LIN {X 0,Y 314.203,Z 248.248,A -85,B 0,C 180,E1 -15768.607,E2 -15768.607} C_VEL
LIN {X 0,Y 312.569,Z 240.551,A -85,B 0,C 180,E1 -15771.085,E2 -15771.085} C_VEL
LIN {X 0,Y 312.557,Z 240.551,A -85,B 0,C 180,E1 -15775.292,E2 -15775.292} C_VEL
LIN {X 0,Y 312.526,Z 240.558,A -85,B 0,C 180,E1 -15778.714,E2 -15778.714} C_VEL
LIN {X 0,Y 312.503,Z 240.561,A -85,B 0,C 180,E1 -15782.666,E2 -15782.666} C_VEL
LIN {X 0,Y 312.507,Z 240.552,A -85,B 0,C 180,E1 -15786.781,E2 -15786.781} C_VEL
LIN {X 0,Y 311.84,Z 240.639,A -85,B 0,C 180,E1 -15787.857,E2 -15787.857} C_VEL
LIN {X 0,Y 308.958,Z 240.997,A -85,B 0,C 180,E1 -15789.608,E2 -15789.608} C_VEL
LIN {X 0,Y 306.532,Z 241.301,A -85,B 0,C 180,E1 -15791.029,E2 -15791.029} C_VEL
LIN {X 0,Y 305.522,Z 241.426,A -85,B 0,C 180,E1 -15792.129,E2 -15792.129} C_VEL
LIN {X 0,Y 305.456,Z 241.437,A -85,B 0,C 180,E1 -15792.502,E2 -15792.502} C_VEL
LIN {X 0,Y 305.443,Z 241.437,A -85,B 0,C 180,E1 -15796.348,E2 -15796.348} C_VEL
LIN {X 0,Y 305.459,Z 241.433,A -85,B 0,C 180,E1 -15799.892,E2 -15799.892} C_VEL
LIN {X 0,Y 305.481,Z 241.43,A -85,B 0,C 180,E1 -15803.632,E2 -15803.632} C_VEL
LIN {X 0,Y 305.466,Z 241.432,A -85,B 0,C 180,E1 -15806.483,E2 -15806.483} C_VEL
LIN {X 0,Y 305.459,Z 241.43,A -85,B 0,C 180,E1 -15809.59,E2 -15809.59} C_VEL
LIN {X 0,Y 305.516,Z 241.431,A -85,B 0,C 180,E1 -15812.608,E2 -15812.608} C_VEL
LIN {X 0,Y 305.509,Z 241.423,A -85,B 0,C 180,E1 -15815.539,E2 -15815.539} C_VEL
LIN {X 0,Y 305.521,Z 241.42,A -85,B 0,C 180,E1 -15819.815,E2 -15819.815} C_VEL
LIN {X 0,Y 305.575,Z 241.422,A -85,B 0,C 180,E1 -15822.603,E2 -15822.603} C_VEL
LIN {X 0,Y 305.65,Z 241.406,A -85,B 0,C 180,E1 -15825.349,E2 -15825.349} C_VEL
LIN {X 0,Y 305.625,Z 241.402,A -85,B 0,C 180,E1 -15829.399,E2 -15829.399} C_VEL
LIN {X 0,Y 305.749,Z 241.393,A -85,B 0,C 180,E1 -15832.073,E2 -15832.073} C_VEL
LIN {X 0,Y 305.674,Z 241.41,A -85,B 0,C 180,E1 -15834.723,E2 -15834.723} C_VEL
LIN {X 0,Y 305.954,Z 241.374,A -85,B 0,C 180,E1 -15838.684,E2 -15838.684} C_VEL
LIN {X 0,Y 305.955,Z 241.371,A -85,B 0,C 180,E1 -15841.316,E2 -15841.316} C_VEL
LIN {X 0,Y 305.853,Z 241.389,A -85,B 0,C 180,E1 -15846.597,E2 -15846.597} C_VEL
LIN {X 0,Y 305.736,Z 241.397,A -85,B 0,C 180,E1 -15849.26,E2 -15849.26} C_VEL
LIN {X 0,Y 305.587,Z 241.416,A -85,B 0,C 180,E1 -15853.296,E2 -15853.296} C_VEL
LIN {X 0,Y 305.551,Z 241.422,A -85,B 0,C 180,E1 -15856.022,E2 -15856.022} C_VEL
LIN {X 0,Y 305.485,Z 241.429,A -85,B 0,C 180,E1 -15860.187,E2 -15860.187} C_VEL
LIN {X 0,Y 305.487,Z 241.432,A -85,B 0,C 180,E1 -15864.463,E2 -15864.463} C_VEL
LIN {X 0,Y 305.467,Z 241.432,A -85,B 0,C 180,E1 -15867.397,E2 -15867.397} C_VEL
LIN {X 0,Y 305.433,Z 241.438,A -85,B 0,C 180,E1 -15870.412,E2 -15870.412} C_VEL
LIN {X 0,Y 305.465,Z 241.434,A -85,B 0,C 180,E1 -15874.078,E2 -15874.078} C_VEL
LIN {X 0,Y 305.469,Z 241.436,A -85,B 0,C 180,E1 -15876.74,E2 -15876.74} C_VEL
LIN {X 0,Y 305.409,Z 241.444,A -85,B 0,C 180,E1 -15880.59,E2 -15880.59} C_VEL
LIN {X 0,Y 305.422,Z 241.438,A -85,B 0,C 180,E1 -15883.656,E2 -15883.656} C_VEL
LIN {X 0,Y 305.454,Z 241.432,A -85,B 0,C 180,E1 -15887.414,E2 -15887.414} C_VEL
LIN {X 0,Y 305.477,Z 241.431,A -85,B 0,C 180,E1 -15891.598,E2 -15891.598} C_VEL
LIN {X 0,Y 305.463,Z 241.436,A -85,B 0,C 180,E1 -15894.887,E2 -15894.887} C_VEL
LIN {X 0,Y 305.481,Z 241.475,A -85,B 0,C 180,E1 -15898.346,E2 -15898.346} C_VEL
LIN {X 0,Y 308.107,Z 253.691,A -85,B 0,C 180,E1 -15902.12,E2 -15902.12} C_VEL
LIN {X 0,Y 309.418,Z 261.563,A -85,B 0,C 180,E1 -15904.434,E2 -15904.434} C_VEL
LIN {X 0,Y 309.266,Z 263.81,A -85,B 0,C 180,E1 -15905.048,E2 -15905.048} C_VEL
LIN {X 0,Y 313.254,Z 289.715,A -85,B 0,C 180,E1 -15905.992,E2 -15905.992} C_VEL
LIN {X 0,Y 315.292,Z 305.062,A -85,B 0,C 180,E1 -15906.504,E2 -15906.504} C_VEL
LIN {X 0,Y 313.764,Z 372.606,A -85,B 0,C 180,E1 -15908.051,E2 -15908.051} C_VEL
LIN {X 0,Y 312.937,Z 386.537,A -85,B 0,C 180,E1 -15908.639,E2 -15908.639} C_VEL
LIN {X 0,Y 311.957,Z 398.459,A -85,B 0,C 180,E1 -15909.39,E2 -15909.39} C_VEL
LIN {X 0,Y 310.802,Z 409.719,A -85,B 0,C 180,E1 -15910.345,E2 -15910.345} C_VEL
LIN {X 0,Y 309.44,Z 421.391,A -85,B 0,C 180,E1 -15911.631,E2 -15911.631} C_VEL
LIN {X 0,Y 308.14,Z 431.519,A -85,B 0,C 180,E1 -15913.036,E2 -15913.036} C_VEL
LIN {X 0,Y 306.995,Z 441.335,A -85,B 0,C 180,E1 -15914.736,E2 -15914.736} C_VEL
LIN {X 0,Y 305.751,Z 450.436,A -85,B 0,C 180,E1 -15916.711,E2 -15916.711} C_VEL
LIN {X 0,Y 304.82,Z 457.766,A -85,B 0,C 180,E1 -15918.698,E2 -15918.698} C_VEL
LIN {X 0,Y 304.223,Z 463.634,A -85,B 0,C 180,E1 -15920.694,E2 -15920.694} C_VEL
LIN {X 0,Y 303.838,Z 468.245,A -85,B 0,C 180,E1 -15922.691,E2 -15922.691} C_VEL
LIN {X 0,Y 303.637,Z 471.745,A -85,B 0,C 180,E1 -15924.688,E2 -15924.688} C_VEL
LIN {X 0,Y 303.633,Z 473.5,A -85,B 0,C 180,E1 -15926.018,E2 -15926.018} C_VEL
LIN {X 0,Y 303.608,Z 474.831,A -85,B 0,C 180,E1 -15927.347,E2 -15927.347} C_VEL
LIN {X 0,Y 303.575,Z 475.764,A -85,B 0,C 180,E1 -15928.673,E2 -15928.673} C_VEL
LIN {X 0,Y 303.604,Z 476.304,A -85,B 0,C 180,E1 -15930,E2 -15930} C_VEL
LIN {X 0,Y 303.565,Z 476.407,A -85,B 0,C 180,E1 -15931.327,E2 -15931.327} C_VEL
LIN {X 0,Y 303.601,Z 476.119,A -85,B 0,C 180,E1 -15932.654,E2 -15932.654} C_VEL
LIN {X 0,Y 303.596,Z 475.445,A -85,B 0,C 180,E1 -15933.982,E2 -15933.982} C_VEL
LIN {X 0,Y 303.695,Z 473.996,A -85,B 0,C 180,E1 -15935.679,E2 -15935.679} C_VEL
LIN {X 0,Y 304.005,Z 470.949,A -85,B 0,C 180,E1 -15937.973,E2 -15937.973} C_VEL
LIN {X 0,Y 304.564,Z 467.224,A -85,B 0,C 180,E1 -15939.966,E2 -15939.966} C_VEL
LIN {X 0,Y 305.367,Z 462.397,A -85,B 0,C 180,E1 -15941.955,E2 -15941.955} C_VEL
LIN {X 0,Y 306.595,Z 456.323,A -85,B 0,C 180,E1 -15943.927,E2 -15943.927} C_VEL
LIN {X 0,Y 308.09,Z 448.786,A -85,B 0,C 180,E1 -15945.887,E2 -15945.887} C_VEL
LIN {X 0,Y 309.541,Z 441.029,A -85,B 0,C 180,E1 -15947.523,E2 -15947.523} C_VEL
LIN {X 0,Y 311.171,Z 431.759,A -85,B 0,C 180,E1 -15949.117,E2 -15949.117} C_VEL
LIN {X 0,Y 313.02,Z 421.391,A -85,B 0,C 180,E1 -15950.537,E2 -15950.537} C_VEL
LIN {X 0,Y 314.798,Z 409.893,A -85,B 0,C 180,E1 -15951.787,E2 -15951.787} C_VEL
LIN {X 0,Y 316.426,Z 397.786,A -85,B 0,C 180,E1 -15952.786,E2 -15952.786} C_VEL
LIN {X 0,Y 317.74,Z 384.331,A -85,B 0,C 180,E1 -15953.591,E2 -15953.591} C_VEL
LIN {X 0,Y 318.583,Z 371.861,A -85,B 0,C 180,E1 -15954.086,E2 -15954.086} C_VEL
LIN {X 0,Y 320.398,Z 307.143,A -85,B 0,C 180,E1 -15955.554,E2 -15955.554} C_VEL
LIN {X 0,Y 317.446,Z 289.422,A -85,B 0,C 180,E1 -15956.282,E2 -15956.282} C_VEL
LIN {X 0,Y 313.767,Z 271.603,A -85,B 0,C 180,E1 -15957.106,E2 -15957.106} C_VEL
LIN {X 0,Y 310.5,Z 263.435,A -85,B 0,C 180,E1 -15957.679,E2 -15957.679} C_VEL
LIN {X 0,Y 308.691,Z 254.815,A -85,B 0,C 180,E1 -15960.435,E2 -15960.435} C_VEL
LIN {X 0,Y 306.228,Z 244.486,A -85,B 0,C 180,E1 -15963.93,E2 -15963.93} C_VEL
LIN {X 0,Y 305.497,Z 241.428,A -85,B 0,C 180,E1 -15965.04,E2 -15965.04} C_VEL
LIN {X 0,Y 305.441,Z 241.438,A -85,B 0,C 180,E1 -15968.527,E2 -15968.527} C_VEL
LIN {X 0,Y 305.455,Z 241.437,A -85,B 0,C 180,E1 -15972.586,E2 -15972.586} C_VEL
LIN {X 0,Y 305.422,Z 241.44,A -85,B 0,C 180,E1 -15976.344,E2 -15976.344} C_VEL
LIN {X 0,Y 305.41,Z 241.442,A -85,B 0,C 180,E1 -15979.885,E2 -15979.885} C_VEL
LIN {X 0,Y 305.463,Z 241.43,A -85,B 0,C 180,E1 -15983.636,E2 -15983.636} C_VEL
LIN {X 0,Y 305.465,Z 241.426,A -85,B 0,C 180,E1 -15986.483,E2 -15986.483} C_VEL
LIN {X 0,Y 305.435,Z 241.433,A -85,B 0,C 180,E1 -15989.588,E2 -15989.588} C_VEL
LIN {X 0,Y 305.472,Z 241.433,A -85,B 0,C 180,E1 -15992.604,E2 -15992.604} C_VEL
LIN {X 0,Y 305.489,Z 241.428,A -85,B 0,C 180,E1 -15995.537,E2 -15995.537} C_VEL
LIN {X 0,Y 305.496,Z 241.428,A -85,B 0,C 180,E1 -15999.814,E2 -15999.814} C_VEL
LIN {X 0,Y 305.545,Z 241.42,A -85,B 0,C 180,E1 -16002.601,E2 -16002.601} C_VEL
LIN {X 0,Y 305.628,Z 241.415,A -85,B 0,C 180,E1 -16005.348,E2 -16005.348} C_VEL
LIN {X 0,Y 305.639,Z 241.408,A -85,B 0,C 180,E1 -16009.4,E2 -16009.4} C_VEL
LIN {X 0,Y 305.81,Z 241.384,A -85,B 0,C 180,E1 -16012.074,E2 -16012.074} C_VEL
LIN {X 0,Y 305.682,Z 241.404,A -85,B 0,C 180,E1 -16014.723,E2 -16014.723} C_VEL
LIN {X 0,Y 305.953,Z 241.364,A -85,B 0,C 180,E1 -16018.684,E2 -16018.684} C_VEL
LIN {X 0,Y 305.954,Z 241.373,A -85,B 0,C 180,E1 -16021.316,E2 -16021.316} C_VEL
LIN {X 0,Y 305.672,Z 241.408,A -85,B 0,C 180,E1 -16025.277,E2 -16025.277} C_VEL
LIN {X 0,Y 305.752,Z 241.388,A -85,B 0,C 180,E1 -16027.927,E2 -16027.927} C_VEL
LIN {X 0,Y 305.6,Z 241.414,A -85,B 0,C 180,E1 -16031.945,E2 -16031.945} C_VEL
LIN {X 0,Y 305.61,Z 241.413,A -85,B 0,C 180,E1 -16035.015,E2 -16035.015} C_VEL
LIN {X 0,Y 305.563,Z 241.418,A -85,B 0,C 180,E1 -16039.437,E2 -16039.437} C_VEL
LIN {X 0,Y 305.492,Z 241.422,A -85,B 0,C 180,E1 -16043.041,E2 -16043.041} C_VEL
LIN {X 0,Y 305.527,Z 241.418,A -85,B 0,C 180,E1 -16046.219,E2 -16046.219} C_VEL
LIN {X 0,Y 305.49,Z 241.432,A -85,B 0,C 180,E1 -16049.048,E2 -16049.048} C_VEL
LIN {X 0,Y 305.444,Z 241.437,A -85,B 0,C 180,E1 -16051.952,E2 -16051.952} C_VEL
LIN {X 0,Y 305.464,Z 241.437,A -85,B 0,C 180,E1 -16055.113,E2 -16055.113} C_VEL
LIN {X 0,Y 305.469,Z 241.433,A -85,B 0,C 180,E1 -16058.533,E2 -16058.533} C_VEL
LIN {X 0,Y 305.46,Z 241.436,A -85,B 0,C 180,E1 -16062.587,E2 -16062.587} C_VEL
LIN {X 0,Y 305.441,Z 241.431,A -85,B 0,C 180,E1 -16066.348,E2 -16066.348} C_VEL
LIN {X 0,Y 305.411,Z 241.44,A -85,B 0,C 180,E1 -16069.885,E2 -16069.885} C_VEL
LIN {X 0,Y 305.486,Z 241.455,A -85,B 0,C 180,E1 -16073.384,E2 -16073.384} C_VEL
LIN {X 0,Y 307.289,Z 248.962,A -85,B 0,C 180,E1 -16076.037,E2 -16076.037} C_VEL
LIN {X 0,Y 315.614,Z 266.974,A -85,B 0,C 180,E1 -16077.391,E2 -16077.391} C_VEL
LIN {X 0,Y 319.918,Z 277.771,A -85,B 0,C 180,E1 -16078.094,E2 -16078.094} C_VEL
LIN {X 0,Y 321.078,Z 283.904,A -85,B 0,C 180,E1 -16078.36,E2 -16078.36} C_VEL
LIN {X 0,Y 318.96,Z 356.614,A -85,B 0,C 180,E1 -16080.007,E2 -16080.007} C_VEL
LIN {X 0,Y 318.074,Z 370.586,A -85,B 0,C 180,E1 -16080.598,E2 -16080.598} C_VEL
LIN {X 0,Y 316.992,Z 382.524,A -85,B 0,C 180,E1 -16081.351,E2 -16081.351} C_VEL
LIN {X 0,Y 315.553,Z 393.762,A -85,B 0,C 180,E1 -16082.294,E2 -16082.294} C_VEL
LIN {X 0,Y 313.929,Z 405.364,A -85,B 0,C 180,E1 -16083.572,E2 -16083.572} C_VEL
LIN {X 0,Y 312.157,Z 415.883,A -85,B 0,C 180,E1 -16085.03,E2 -16085.03} C_VEL
LIN {X 0,Y 310.4,Z 425.242,A -85,B 0,C 180,E1 -16086.657,E2 -16086.657} C_VEL
LIN {X 0,Y 308.671,Z 434.282,A -85,B 0,C 180,E1 -16088.636,E2 -16088.636} C_VEL
LIN {X 0,Y 307.202,Z 441.538,A -85,B 0,C 180,E1 -16090.627,E2 -16090.627} C_VEL
LIN {X 0,Y 305.99,Z 447.301,A -85,B 0,C 180,E1 -16092.627,E2 -16092.627} C_VEL
LIN {X 0,Y 305.111,Z 451.814,A -85,B 0,C 180,E1 -16094.639,E2 -16094.639} C_VEL
LIN {X 0,Y 304.426,Z 455.23,A -85,B 0,C 180,E1 -16096.652,E2 -16096.652} C_VEL
LIN {X 0,Y 304.065,Z 456.919,A -85,B 0,C 180,E1 -16097.994,E2 -16097.994} C_VEL
LIN {X 0,Y 303.653,Z 459.087,A -85,B 0,C 180,E1 -16100.676,E2 -16100.676} C_VEL
LIN {X 0,Y 303.619,Z 459.549,A -85,B 0,C 180,E1 -16102.017,E2 -16102.017} C_VEL
LIN {X 0,Y 303.622,Z 459.352,A -85,B 0,C 180,E1 -16104.464,E2 -16104.464} C_VEL
LIN {X 0,Y 303.648,Z 458.56,A -85,B 0,C 180,E1 -16106.018,E2 -16106.018} C_VEL
LIN {X 0,Y 303.661,Z 457.434,A -85,B 0,C 180,E1 -16107.347,E2 -16107.347} C_VEL
LIN {X 0,Y 303.935,Z 453.917,A -85,B 0,C 180,E1 -16110,E2 -16110} C_VEL
LIN {X 0,Y 304.323,Z 450.115,A -85,B 0,C 180,E1 -16111.985,E2 -16111.985} C_VEL
LIN {X 0,Y 304.901,Z 445.198,A -85,B 0,C 180,E1 -16113.965,E2 -16113.965} C_VEL
LIN {X 0,Y 305.66,Z 439.023,A -85,B 0,C 180,E1 -16115.939,E2 -16115.939} C_VEL
LIN {X 0,Y 306.784,Z 431.306,A -85,B 0,C 180,E1 -16117.9,E2 -16117.9} C_VEL
LIN {X 0,Y 308.173,Z 421.655,A -85,B 0,C 180,E1 -16119.848,E2 -16119.848} C_VEL
LIN {X 0,Y 309.434,Z 411.687,A -85,B 0,C 180,E1 -16121.463,E2 -16121.463} C_VEL
LIN {X 0,Y 310.732,Z 400.394,A -85,B 0,C 180,E1 -16122.906,E2 -16122.906} C_VEL
LIN {X 0,Y 311.868,Z 389.33,A -85,B 0,C 180,E1 -16124.02,E2 -16124.02} C_VEL
LIN {X 0,Y 312.948,Z 376.702,A -85,B 0,C 180,E1 -16124.986,E2 -16124.986} C_VEL
LIN {X 0,Y 313.662,Z 363.863,A -85,B 0,C 180,E1 -16125.681,E2 -16125.681} C_VEL
LIN {X 0,Y 314.124,Z 351.155,A -85,B 0,C 180,E1 -16126.115,E2 -16126.115} C_VEL
LIN {X 0,Y 315.815,Z 279.626,A -85,B 0,C 180,E1 -16127.715,E2 -16127.715} C_VEL
LIN {X 0,Y 312.921,Z 264.379,A -85,B 0,C 180,E1 -16128.293,E2 -16128.293} C_VEL
LIN {X 0,Y 307.038,Z 248.411,A -85,B 0,C 180,E1 -16129.163,E2 -16129.163} C_VEL
LIN {X 0,Y 305.523,Z 241.427,A -85,B 0,C 180,E1 -16131.507,E2 -16131.507} C_VEL
LIN {X 0,Y 305.51,Z 241.428,A -85,B 0,C 180,E1 -16135.918,E2 -16135.918} C_VEL
LIN {X 0,Y 305.465,Z 241.435,A -85,B 0,C 180,E1 -16139.039,E2 -16139.039} C_VEL
LIN {X 0,Y 305.439,Z 241.436,A -85,B 0,C 180,E1 -16141.953,E2 -16141.953} C_VEL
LIN {X 0,Y 305.464,Z 241.434,A -85,B 0,C 180,E1 -16145.113,E2 -16145.113} C_VEL
LIN {X 0,Y 305.451,Z 241.438,A -85,B 0,C 180,E1 -16148.529,E2 -16148.529} C_VEL
LIN {X 0,Y 305.456,Z 241.437,A -85,B 0,C 180,E1 -16152.502,E2 -16152.502} C_VEL
LIN {X 0,Y 304.819,Z 241.522,A -85,B 0,C 180,E1 -16153.601,E2 -16153.601} C_VEL
LIN {X 0,Y 301.929,Z 241.878,A -85,B 0,C 180,E1 -16155.388,E2 -16155.388} C_VEL
LIN {X 0,Y 299.469,Z 242.183,A -85,B 0,C 180,E1 -16156.839,E2 -16156.839} C_VEL
LIN {X 0,Y 298.435,Z 242.308,A -85,B 0,C 180,E1 -16157.963,E2 -16157.963} C_VEL
LIN {X 0,Y 298.365,Z 242.318,A -85,B 0,C 180,E1 -16158.344,E2 -16158.344} C_VEL
LIN {X 0,Y 298.409,Z 242.312,A -85,B 0,C 180,E1 -16162.241,E2 -16162.241} C_VEL
LIN {X 0,Y 298.409,Z 242.309,A -85,B 0,C 180,E1 -16165.581,E2 -16165.581} C_VEL
LIN {X 0,Y 298.393,Z 242.31,A -85,B 0,C 180,E1 -16168.791,E2 -16168.791} C_VEL
LIN {X 0,Y 298.458,Z 242.305,A -85,B 0,C 180,E1 -16171.903,E2 -16171.903} C_VEL
LIN {X 0,Y 298.484,Z 242.3,A -85,B 0,C 180,E1 -16174.924,E2 -16174.924} C_VEL
LIN {X 0,Y 298.451,Z 242.301,A -85,B 0,C 180,E1 -16179.315,E2 -16179.315} C_VEL
LIN {X 0,Y 298.539,Z 242.295,A -85,B 0,C 180,E1 -16182.179,E2 -16182.179} C_VEL
LIN {X 0,Y 298.594,Z 242.286,A -85,B 0,C 180,E1 -16184.995,E2 -16184.995} C_VEL
LIN {X 0,Y 298.584,Z 242.279,A -85,B 0,C 180,E1 -16189.146,E2 -16189.146} C_VEL
LIN {X 0,Y 298.7,Z 242.27,A -85,B 0,C 180,E1 -16191.884,E2 -16191.884} C_VEL
LIN {X 0,Y 298.642,Z 242.286,A -85,B 0,C 180,E1 -16194.598,E2 -16194.598} C_VEL
LIN {X 0,Y 298.921,Z 242.249,A -85,B 0,C 180,E1 -16198.653,E2 -16198.653} C_VEL
LIN {X 0,Y 298.922,Z 242.247,A -85,B 0,C 180,E1 -16201.347,E2 -16201.347} C_VEL
LIN {X 0,Y 298.798,Z 242.267,A -85,B 0,C 180,E1 -16206.754,E2 -16206.754} C_VEL
LIN {X 0,Y 298.681,Z 242.275,A -85,B 0,C 180,E1 -16209.48,E2 -16209.48} C_VEL
LIN {X 0,Y 298.546,Z 242.293,A -85,B 0,C 180,E1 -16213.616,E2 -16213.616} C_VEL
LIN {X 0,Y 298.484,Z 242.305,A -85,B 0,C 180,E1 -16216.412,E2 -16216.412} C_VEL
LIN {X 0,Y 298.46,Z 242.302,A -85,B 0,C 180,E1 -16219.627,E2 -16219.627} C_VEL
LIN {X 0,Y 298.424,Z 242.308,A -85,B 0,C 180,E1 -16223.6,E2 -16223.6} C_VEL
LIN {X 0,Y 298.413,Z 242.314,A -85,B 0,C 180,E1 -16226.582,E2 -16226.582} C_VEL
LIN {X 0,Y 298.398,Z 242.311,A -85,B 0,C 180,E1 -16229.643,E2 -16229.643} C_VEL
LIN {X 0,Y 298.392,Z 242.316,A -85,B 0,C 180,E1 -16232.801,E2 -16232.801} C_VEL
LIN {X 0,Y 298.442,Z 242.31,A -85,B 0,C 180,E1 -16236.806,E2 -16236.806} C_VEL
LIN {X 0,Y 298.348,Z 242.32,A -85,B 0,C 180,E1 -16241.079,E2 -16241.079} C_VEL
LIN {X 0,Y 298.399,Z 242.314,A -85,B 0,C 180,E1 -16243.103,E2 -16243.103} C_VEL
LIN {X 0,Y 298.403,Z 242.312,A -85,B 0,C 180,E1 -16246.921,E2 -16246.921} C_VEL
LIN {X 0,Y 298.404,Z 242.313,A -85,B 0,C 180,E1 -16251.006,E2 -16251.006} C_VEL
LIN {X 0,Y 298.433,Z 242.31,A -85,B 0,C 180,E1 -16253.932,E2 -16253.932} C_VEL
LIN {X 0,Y 298.433,Z 242.519,A -85,B 0,C 180,E1 -16257.972,E2 -16257.972} C_VEL
LIN {X 0,Y 300.775,Z 253.216,A -85,B 0,C 180,E1 -16261.379,E2 -16261.379} C_VEL
LIN {X 0,Y 302.428,Z 262.577,A -85,B 0,C 180,E1 -16264.216,E2 -16264.216} C_VEL
LIN {X 0,Y 302.48,Z 263.631,A -85,B 0,C 180,E1 -16264.521,E2 -16264.521} C_VEL
LIN {X 0,Y 306.547,Z 289.629,A -85,B 0,C 180,E1 -16265.498,E2 -16265.498} C_VEL
LIN {X 0,Y 308.645,Z 305.97,A -85,B 0,C 180,E1 -16266.055,E2 -16266.055} C_VEL
LIN {X 0,Y 307.12,Z 371.987,A -85,B 0,C 180,E1 -16267.595,E2 -16267.595} C_VEL
LIN {X 0,Y 306.318,Z 385.292,A -85,B 0,C 180,E1 -16268.154,E2 -16268.154} C_VEL
LIN {X 0,Y 305.322,Z 397.489,A -85,B 0,C 180,E1 -16268.921,E2 -16268.921} C_VEL
LIN {X 0,Y 304.095,Z 408.965,A -85,B 0,C 180,E1 -16269.893,E2 -16269.893} C_VEL
LIN {X 0,Y 302.674,Z 420.748,A -85,B 0,C 180,E1 -16271.206,E2 -16271.206} C_VEL
LIN {X 0,Y 301.271,Z 431.211,A -85,B 0,C 180,E1 -16272.679,E2 -16272.679} C_VEL
LIN {X 0,Y 300.124,Z 440.854,A -85,B 0,C 180,E1 -16274.378,E2 -16274.378} C_VEL
LIN {X 0,Y 298.819,Z 450.007,A -85,B 0,C 180,E1 -16276.397,E2 -16276.397} C_VEL
LIN {X 0,Y 297.807,Z 457.377,A -85,B 0,C 180,E1 -16278.428,E2 -16278.428} C_VEL
LIN {X 0,Y 297.195,Z 463.286,A -85,B 0,C 180,E1 -16280.472,E2 -16280.472} C_VEL
LIN {X 0,Y 296.785,Z 467.932,A -85,B 0,C 180,E1 -16282.516,E2 -16282.516} C_VEL
LIN {X 0,Y 296.552,Z 471.46,A -85,B 0,C 180,E1 -16284.56,E2 -16284.56} C_VEL
LIN {X 0,Y 296.531,Z 473.241,A -85,B 0,C 180,E1 -16285.923,E2 -16285.923} C_VEL
LIN {X 0,Y 296.534,Z 474.588,A -85,B 0,C 180,E1 -16287.283,E2 -16287.283} C_VEL
LIN {X 0,Y 296.494,Z 475.534,A -85,B 0,C 180,E1 -16288.642,E2 -16288.642} C_VEL
LIN {X 0,Y 296.518,Z 476.092,A -85,B 0,C 180,E1 -16290,E2 -16290} C_VEL
LIN {X 0,Y 296.485,Z 476.218,A -85,B 0,C 180,E1 -16291.358,E2 -16291.358} C_VEL
LIN {X 0,Y 296.526,Z 475.943,A -85,B 0,C 180,E1 -16292.717,E2 -16292.717} C_VEL
LIN {X 0,Y 296.554,Z 474.235,A -85,B 0,C 180,E1 -16295.44,E2 -16295.44} C_VEL
LIN {X 0,Y 296.694,Z 472.757,A -85,B 0,C 180,E1 -16296.802,E2 -16296.802} C_VEL
LIN {X 0,Y 297.109,Z 469.75,A -85,B 0,C 180,E1 -16298.845,E2 -16298.845} C_VEL
LIN {X 0,Y 297.806,Z 465.703,A -85,B 0,C 180,E1 -16300.882,E2 -16300.882} C_VEL
LIN {X 0,Y 298.943,Z 459.502,A -85,B 0,C 180,E1 -16303.251,E2 -16303.251} C_VEL
LIN {X 0,Y 300.491,Z 452.767,A -85,B 0,C 180,E1 -16305.255,E2 -16305.255} C_VEL
LIN {X 0,Y 302.131,Z 444.475,A -85,B 0,C 180,E1 -16307.241,E2 -16307.241} C_VEL
LIN {X 0,Y 303.7,Z 435.852,A -85,B 0,C 180,E1 -16308.904,E2 -16308.904} C_VEL
LIN {X 0,Y 305.745,Z 425.298,A -85,B 0,C 180,E1 -16310.521,E2 -16310.521} C_VEL
LIN {X 0,Y 307.497,Z 414.847,A -85,B 0,C 180,E1 -16311.802,E2 -16311.802} C_VEL
LIN {X 0,Y 309.257,Z 403.325,A -85,B 0,C 180,E1 -16312.903,E2 -16312.903} C_VEL
LIN {X 0,Y 310.698,Z 391.377,A -85,B 0,C 180,E1 -16313.761,E2 -16313.761} C_VEL
LIN {X 0,Y 311.845,Z 378.463,A -85,B 0,C 180,E1 -16314.419,E2 -16314.419} C_VEL
LIN {X 0,Y 312.563,Z 366.37,A -85,B 0,C 180,E1 -16314.802,E2 -16314.802} C_VEL
LIN {X 0,Y 314.036,Z 306.607,A -85,B 0,C 180,E1 -16316.181,E2 -16316.181} C_VEL
LIN {X 0,Y 309.092,Z 279.498,A -85,B 0,C 180,E1 -16317.388,E2 -16317.388} C_VEL
LIN {X 0,Y 307.454,Z 273.208,A -85,B 0,C 180,E1 -16317.728,E2 -16317.728} C_VEL
LIN {X 0,Y 303.263,Z 263.264,A -85,B 0,C 180,E1 -16318.458,E2 -16318.458} C_VEL
LIN {X 0,Y 301.198,Z 253.595,A -85,B 0,C 180,E1 -16321.669,E2 -16321.669} C_VEL
LIN {X 0,Y 298.447,Z 242.339,A -85,B 0,C 180,E1 -16325.667,E2 -16325.667} C_VEL
LIN {X 0,Y 298.401,Z 242.316,A -85,B 0,C 180,E1 -16329.487,E2 -16329.487} C_VEL
LIN {X 0,Y 298.399,Z 242.316,A -85,B 0,C 180,E1 -16333.103,E2 -16333.103} C_VEL
LIN {X 0,Y 298.372,Z 242.32,A -85,B 0,C 180,E1 -16336.915,E2 -16336.915} C_VEL
LIN {X 0,Y 298.385,Z 242.316,A -85,B 0,C 180,E1 -16341.011,E2 -16341.011} C_VEL
LIN {X 0,Y 298.405,Z 242.311,A -85,B 0,C 180,E1 -16343.928,E2 -16343.928} C_VEL
LIN {X 0,Y 298.393,Z 242.308,A -85,B 0,C 180,E1 -16347.2,E2 -16347.2} C_VEL
LIN {X 0,Y 298.411,Z 242.303,A -85,B 0,C 180,E1 -16350.622,E2 -16350.622} C_VEL
LIN {X 0,Y 298.45,Z 242.3,A -85,B 0,C 180,E1 -16354.921,E2 -16354.921} C_VEL
LIN {X 0,Y 298.43,Z 242.304,A -85,B 0,C 180,E1 -16359.314,E2 -16359.314} C_VEL
LIN {X 0,Y 298.506,Z 242.297,A -85,B 0,C 180,E1 -16362.177,E2 -16362.177} C_VEL
LIN {X 0,Y 298.586,Z 242.289,A -85,B 0,C 180,E1 -16364.994,E2 -16364.994} C_VEL
LIN {X 0,Y 298.594,Z 242.283,A -85,B 0,C 180,E1 -16369.147,E2 -16369.147} C_VEL
LIN {X 0,Y 298.756,Z 242.263,A -85,B 0,C 180,E1 -16371.886,E2 -16371.886} C_VEL
LIN {X 0,Y 298.653,Z 242.279,A -85,B 0,C 180,E1 -16374.599,E2 -16374.599} C_VEL
LIN {X 0,Y 298.919,Z 242.24,A -85,B 0,C 180,E1 -16378.653,E2 -16378.653} C_VEL
LIN {X 0,Y 298.921,Z 242.248,A -85,B 0,C 180,E1 -16381.347,E2 -16381.347} C_VEL
LIN {X 0,Y 298.712,Z 242.273,A -85,B 0,C 180,E1 -16386.513,E2 -16386.513} C_VEL
LIN {X 0,Y 298.627,Z 242.281,A -85,B 0,C 180,E1 -16389.482,E2 -16389.482} C_VEL
LIN {X 0,Y 298.546,Z 242.287,A -85,B 0,C 180,E1 -16393.616,E2 -16393.616} C_VEL
LIN {X 0,Y 298.488,Z 242.301,A -85,B 0,C 180,E1 -16396.412,E2 -16396.412} C_VEL
LIN {X 0,Y 298.5,Z 242.3,A -85,B 0,C 180,E1 -16399.648,E2 -16399.648} C_VEL
LIN {X 0,Y 298.459,Z 242.303,A -85,B 0,C 180,E1 -16403.598,E2 -16403.598} C_VEL
LIN {X 0,Y 298.486,Z 242.294,A -85,B 0,C 180,E1 -16406.575,E2 -16406.575} C_VEL
LIN {X 0,Y 298.418,Z 242.307,A -85,B 0,C 180,E1 -16409.642,E2 -16409.642} C_VEL
LIN {X 0,Y 298.396,Z 242.314,A -85,B 0,C 180,E1 -16412.8,E2 -16412.8} C_VEL
LIN {X 0,Y 298.466,Z 242.302,A -85,B 0,C 180,E1 -16416.812,E2 -16416.812} C_VEL
LIN {X 0,Y 298.389,Z 242.315,A -85,B 0,C 180,E1 -16421.088,E2 -16421.088} C_VEL
LIN {X 0,Y 298.39,Z 242.32,A -85,B 0,C 180,E1 -16425.042,E2 -16425.042} C_VEL
LIN {X 0,Y 298.351,Z 242.328,A -85,B 0,C 180,E1 -16428.733,E2 -16428.733} C_VEL
LIN {X 0,Y 298.452,Z 242.491,A -85,B 0,C 180,E1 -16432.778,E2 -16432.778} C_VEL
LIN {X 0,Y 300.129,Z 249.165,A -85,B 0,C 180,E1 -16435.227,E2 -16435.227} C_VEL
LIN {X 0,Y 309.605,Z 269.427,A -85,B 0,C 180,E1 -16436.829,E2 -16436.829} C_VEL
LIN {X 0,Y 313.908,Z 280.009,A -85,B 0,C 180,E1 -16437.552,E2 -16437.552} C_VEL
LIN {X 0,Y 314.781,Z 284.041,A -85,B 0,C 180,E1 -16437.744,E2 -16437.744} C_VEL
LIN {X 0,Y 312.631,Z 356.824,A -85,B 0,C 180,E1 -16439.428,E2 -16439.428} C_VEL
LIN {X 0,Y 311.72,Z 370.794,A -85,B 0,C 180,E1 -16440.031,E2 -16440.031} C_VEL
LIN {X 0,Y 310.575,Z 382.725,A -85,B 0,C 180,E1 -16440.795,E2 -16440.795} C_VEL
LIN {X 0,Y 308.994,Z 394.764,A -85,B 0,C 180,E1 -16441.839,E2 -16441.839} C_VEL
LIN {X 0,Y 307.329,Z 405.969,A -85,B 0,C 180,E1 -16443.108,E2 -16443.108} C_VEL
LIN {X 0,Y 305.445,Z 416.607,A -85,B 0,C 180,E1 -16444.625,E2 -16444.625} C_VEL
LIN {X 0,Y 303.783,Z 425.029,A -85,B 0,C 180,E1 -16446.118,E2 -16446.118} C_VEL
LIN {X 0,Y 301.949,Z 434.139,A -85,B 0,C 180,E1 -16448.136,E2 -16448.136} C_VEL
LIN {X 0,Y 300.395,Z 441.456,A -85,B 0,C 180,E1 -16450.169,E2 -16450.169} C_VEL
LIN {X 0,Y 299.111,Z 447.287,A -85,B 0,C 180,E1 -16452.215,E2 -16452.215} C_VEL
LIN {X 0,Y 298.166,Z 451.853,A -85,B 0,C 180,E1 -16454.272,E2 -16454.272} C_VEL
LIN {X 0,Y 297.44,Z 455.31,A -85,B 0,C 180,E1 -16456.333,E2 -16456.333} C_VEL
LIN {X 0,Y 297.051,Z 457.026,A -85,B 0,C 180,E1 -16457.706,E2 -16457.706} C_VEL
LIN {X 0,Y 296.573,Z 459.235,A -85,B 0,C 180,E1 -16460.451,E2 -16460.451} C_VEL
LIN {X 0,Y 296.524,Z 459.736,A -85,B 0,C 180,E1 -16461.824,E2 -16461.824} C_VEL
LIN {X 0,Y 296.548,Z 459.522,A -85,B 0,C 180,E1 -16464.491,E2 -16464.491} C_VEL
LIN {X 0,Y 296.542,Z 458.807,A -85,B 0,C 180,E1 -16465.923,E2 -16465.923} C_VEL
LIN {X 0,Y 296.583,Z 457.718,A -85,B 0,C 180,E1 -16467.284,E2 -16467.284} C_VEL
LIN {X 0,Y 296.834,Z 454.246,A -85,B 0,C 180,E1 -16470,E2 -16470} C_VEL
LIN {X 0,Y 297.261,Z 450.487,A -85,B 0,C 180,E1 -16472.032,E2 -16472.032} C_VEL
LIN {X 0,Y 297.841,Z 445.618,A -85,B 0,C 180,E1 -16474.059,E2 -16474.059} C_VEL
LIN {X 0,Y 298.64,Z 439.493,A -85,B 0,C 180,E1 -16476.079,E2 -16476.079} C_VEL
LIN {X 0,Y 299.772,Z 431.868,A -85,B 0,C 180,E1 -16478.086,E2 -16478.086} C_VEL
LIN {X 0,Y 301.214,Z 422.29,A -85,B 0,C 180,E1 -16480.078,E2 -16480.078} C_VEL
LIN {X 0,Y 302.506,Z 412.426,A -85,B 0,C 180,E1 -16481.729,E2 -16481.729} C_VEL
LIN {X 0,Y 303.877,Z 401.291,A -85,B 0,C 180,E1 -16483.202,E2 -16483.202} C_VEL
LIN {X 0,Y 305.031,Z 390.396,A -85,B 0,C 180,E1 -16484.34,E2 -16484.34} C_VEL
LIN {X 0,Y 306.165,Z 378.076,A -85,B 0,C 180,E1 -16485.326,E2 -16485.326} C_VEL
LIN {X 0,Y 306.92,Z 364.959,A -85,B 0,C 180,E1 -16486.077,E2 -16486.077} C_VEL
LIN {X 0,Y 307.423,Z 352.82,A -85,B 0,C 180,E1 -16486.519,E2 -16486.519} C_VEL
LIN {X 0,Y 309.104,Z 279.856,A -85,B 0,C 180,E1 -16488.198,E2 -16488.198} C_VEL
LIN {X 0,Y 306.686,Z 267.023,A -85,B 0,C 180,E1 -16488.699,E2 -16488.699} C_VEL
LIN {X 0,Y 299.865,Z 248.66,A -85,B 0,C 180,E1 -16489.724,E2 -16489.724} C_VEL
LIN {X 0,Y 298.441,Z 242.309,A -85,B 0,C 180,E1 -16491.862,E2 -16491.862} C_VEL
LIN {X 0,Y 298.452,Z 242.309,A -85,B 0,C 180,E1 -16495.079,E2 -16495.079} C_VEL
LIN {X 0,Y 298.412,Z 242.312,A -85,B 0,C 180,E1 -16499.378,E2 -16499.378} C_VEL
LIN {X 0,Y 298.394,Z 242.317,A -85,B 0,C 180,E1 -16502.8,E2 -16502.8} C_VEL
LIN {X 0,Y 298.448,Z 242.31,A -85,B 0,C 180,E1 -16506.807,E2 -16506.807} C_VEL
LIN {X 0,Y 298.389,Z 242.315,A -85,B 0,C 180,E1 -16511.088,E2 -16511.088} C_VEL
LIN {X 0,Y 298.39,Z 242.316,A -85,B 0,C 180,E1 -16515.041,E2 -16515.041} C_VEL
LIN {X 0,Y 298.365,Z 242.318,A -85,B 0,C 180,E1 -16518.344,E2 -16518.344} C_VEL
LIN {X 0,Y 297.729,Z 242.401,A -85,B 0,C 180,E1 -16519.47,E2 -16519.47} C_VEL
LIN {X 0,Y 294.877,Z 242.754,A -85,B 0,C 180,E1 -16521.304,E2 -16521.304} C_VEL
LIN {X 0,Y 292.45,Z 243.058,A -85,B 0,C 180,E1 -16522.792,E2 -16522.792} C_VEL
LIN {X 0,Y 291.424,Z 243.182,A -85,B 0,C 180,E1 -16523.945,E2 -16523.945} C_VEL
LIN {X 0,Y 291.351,Z 243.191,A -85,B 0,C 180,E1 -16524.335,E2 -16524.335} C_VEL
LIN {X 0,Y 291.371,Z 243.178,A -85,B 0,C 180,E1 -16527.95,E2 -16527.95} C_VEL
LIN {X 0,Y 291.378,Z 243.188,A -85,B 0,C 180,E1 -16531.158,E2 -16531.158} C_VEL
LIN {X 0,Y 291.414,Z 243.184,A -85,B 0,C 180,E1 -16534.271,E2 -16534.271} C_VEL
LIN {X 0,Y 291.382,Z 243.173,A -85,B 0,C 180,E1 -16537.299,E2 -16537.299} C_VEL
LIN {X 0,Y 291.459,Z 243.173,A -85,B 0,C 180,E1 -16540.27,E2 -16540.27} C_VEL
LIN {X 0,Y 291.556,Z 243.166,A -85,B 0,C 180,E1 -16544.624,E2 -16544.624} C_VEL
LIN {X 0,Y 291.53,Z 243.156,A -85,B 0,C 180,E1 -16548.88,E2 -16548.88} C_VEL
LIN {X 0,Y 291.653,Z 243.147,A -85,B 0,C 180,E1 -16551.687,E2 -16551.687} C_VEL
LIN {X 0,Y 291.61,Z 243.16,A -85,B 0,C 180,E1 -16554.468,E2 -16554.468} C_VEL
LIN {X 0,Y 291.888,Z 243.124,A -85,B 0,C 180,E1 -16558.62,E2 -16558.62} C_VEL
LIN {X 0,Y 291.888,Z 243.123,A -85,B 0,C 180,E1 -16561.38,E2 -16561.38} C_VEL
LIN {X 0,Y 291.747,Z 243.144,A -85,B 0,C 180,E1 -16566.918,E2 -16566.918} C_VEL
LIN {X 0,Y 291.63,Z 243.153,A -85,B 0,C 180,E1 -16569.712,E2 -16569.712} C_VEL
LIN {X 0,Y 291.516,Z 243.17,A -85,B 0,C 180,E1 -16573.95,E2 -16573.95} C_VEL
LIN {X 0,Y 291.429,Z 243.181,A -85,B 0,C 180,E1 -16576.821,E2 -16576.821} C_VEL
LIN {X 0,Y 291.424,Z 243.179,A -85,B 0,C 180,E1 -16579.86,E2 -16579.86} C_VEL
LIN {X 0,Y 291.365,Z 243.189,A -85,B 0,C 180,E1 -16584.208,E2 -16584.208} C_VEL
LIN {X 0,Y 291.359,Z 243.19,A -85,B 0,C 180,E1 -16587.278,E2 -16587.278} C_VEL
LIN {X 0,Y 291.32,Z 243.195,A -85,B 0,C 180,E1 -16590.439,E2 -16590.439} C_VEL
LIN {X 0,Y 291.344,Z 243.191,A -85,B 0,C 180,E1 -16593.698,E2 -16593.698} C_VEL
LIN {X 0,Y 291.368,Z 243.189,A -85,B 0,C 180,E1 -16597.252,E2 -16597.252} C_VEL
LIN {X 0,Y 291.3,Z 243.201,A -85,B 0,C 180,E1 -16600.648,E2 -16600.648} C_VEL
LIN {X 0,Y 291.291,Z 243.202,A -85,B 0,C 180,E1 -16604.402,E2 -16604.402} C_VEL
LIN {X 0,Y 291.326,Z 243.192,A -85,B 0,C 180,E1 -16608.404,E2 -16608.404} C_VEL
LIN {X 0,Y 291.354,Z 243.191,A -85,B 0,C 180,E1 -16611.159,E2 -16611.159} C_VEL
LIN {X 0,Y 291.386,Z 243.191,A -85,B 0,C 180,E1 -16614.63,E2 -16614.63} C_VEL
LIN {X 0,Y 291.364,Z 243.198,A -85,B 0,C 180,E1 -16617.462,E2 -16617.462} C_VEL
LIN {X 0,Y 293.74,Z 254.053,A -85,B 0,C 180,E1 -16621.02,E2 -16621.02} C_VEL
LIN {X 0,Y 295.446,Z 263.563,A -85,B 0,C 180,E1 -16623.958,E2 -16623.958} C_VEL
LIN {X 0,Y 296.941,Z 270.938,A -85,B 0,C 180,E1 -16624.272,E2 -16624.272} C_VEL
LIN {X 0,Y 301.135,Z 299.015,A -85,B 0,C 180,E1 -16625.322,E2 -16625.322} C_VEL
LIN {X 0,Y 302.03,Z 307.217,A -85,B 0,C 180,E1 -16625.596,E2 -16625.596} C_VEL
LIN {X 0,Y 300.434,Z 372.513,A -85,B 0,C 180,E1 -16627.159,E2 -16627.159} C_VEL
LIN {X 0,Y 299.552,Z 386.345,A -85,B 0,C 180,E1 -16627.77,E2 -16627.77} C_VEL
LIN {X 0,Y 298.45,Z 398.742,A -85,B 0,C 180,E1 -16628.593,E2 -16628.593} C_VEL
LIN {X 0,Y 296.998,Z 411.417,A -85,B 0,C 180,E1 -16629.752,E2 -16629.752} C_VEL
LIN {X 0,Y 295.556,Z 422.706,A -85,B 0,C 180,E1 -16631.096,E2 -16631.096} C_VEL
LIN {X 0,Y 294.187,Z 432.859,A -85,B 0,C 180,E1 -16632.626,E2 -16632.626} C_VEL
LIN {X 0,Y 292.994,Z 442.021,A -85,B 0,C 180,E1 -16634.345,E2 -16634.345} C_VEL
LIN {X 0,Y 291.678,Z 450.942,A -85,B 0,C 180,E1 -16636.413,E2 -16636.413} C_VEL
LIN {X 0,Y 290.687,Z 458.093,A -85,B 0,C 180,E1 -16638.495,E2 -16638.495} C_VEL
LIN {X 0,Y 289.989,Z 464.607,A -85,B 0,C 180,E1 -16640.936,E2 -16640.936} C_VEL
LIN {X 0,Y 289.606,Z 468.899,A -85,B 0,C 180,E1 -16643.031,E2 -16643.031} C_VEL
LIN {X 0,Y 289.479,Z 471.292,A -85,B 0,C 180,E1 -16644.505,E2 -16644.505} C_VEL
LIN {X 0,Y 289.432,Z 472.982,A -85,B 0,C 180,E1 -16645.823,E2 -16645.823} C_VEL
LIN {X 0,Y 289.439,Z 474.343,A -85,B 0,C 180,E1 -16647.217,E2 -16647.217} C_VEL
LIN {X 0,Y 289.416,Z 475.304,A -85,B 0,C 180,E1 -16648.609,E2 -16648.609} C_VEL
LIN {X 0,Y 289.436,Z 475.876,A -85,B 0,C 180,E1 -16650,E2 -16650} C_VEL
LIN {X 0,Y 289.407,Z 476.029,A -85,B 0,C 180,E1 -16651.392,E2 -16651.392} C_VEL
LIN {X 0,Y 289.43,Z 475.766,A -85,B 0,C 180,E1 -16652.784,E2 -16652.784} C_VEL
LIN {X 0,Y 289.48,Z 474.086,A -85,B 0,C 180,E1 -16655.573,E2 -16655.573} C_VEL
LIN {X 0,Y 289.639,Z 472.637,A -85,B 0,C 180,E1 -16656.969,E2 -16656.969} C_VEL
LIN {X 0,Y 290.073,Z 469.654,A -85,B 0,C 180,E1 -16659.061,E2 -16659.061} C_VEL
LIN {X 0,Y 290.815,Z 465.637,A -85,B 0,C 180,E1 -16661.147,E2 -16661.147} C_VEL
LIN {X 0,Y 292.026,Z 459.478,A -85,B 0,C 180,E1 -16663.571,E2 -16663.571} C_VEL
LIN {X 0,Y 293.648,Z 452.781,A -85,B 0,C 180,E1 -16665.62,E2 -16665.62} C_VEL
LIN {X 0,Y 295.433,Z 444.187,A -85,B 0,C 180,E1 -16667.727,E2 -16667.727} C_VEL
LIN {X 0,Y 296.989,Z 435.988,A -85,B 0,C 180,E1 -16669.348,E2 -16669.348} C_VEL
LIN {X 0,Y 299.125,Z 425.502,A -85,B 0,C 180,E1 -16670.996,E2 -16670.996} C_VEL
LIN {X 0,Y 301.19,Z 413.713,A -85,B 0,C 180,E1 -16672.464,E2 -16672.464} C_VEL
LIN {X 0,Y 303.029,Z 401.832,A -85,B 0,C 180,E1 -16673.583,E2 -16673.583} C_VEL
LIN {X 0,Y 304.531,Z 389.485,A -85,B 0,C 180,E1 -16674.454,E2 -16674.454} C_VEL
LIN {X 0,Y 305.669,Z 376.783,A -85,B 0,C 180,E1 -16675.082,E2 -16675.082} C_VEL
LIN {X 0,Y 306.338,Z 363.425,A -85,B 0,C 180,E1 -16675.478,E2 -16675.478} C_VEL
LIN {X 0,Y 307.776,Z 307.826,A -85,B 0,C 180,E1 -16676.783,E2 -16676.783} C_VEL
LIN {X 0,Y 303.206,Z 282.053,A -85,B 0,C 180,E1 -16677.955,E2 -16677.955} C_VEL
LIN {X 0,Y 301.803,Z 276.442,A -85,B 0,C 180,E1 -16678.263,E2 -16678.263} C_VEL
LIN {X 0,Y 296.056,Z 262.898,A -85,B 0,C 180,E1 -16679.34,E2 -16679.34} C_VEL
LIN {X 0,Y 293.593,Z 252.105,A -85,B 0,C 180,E1 -16683.089,E2 -16683.089} C_VEL
LIN {X 0,Y 291.407,Z 243.186,A -85,B 0,C 180,E1 -16686.434,E2 -16686.434} C_VEL
LIN {X 0,Y 291.333,Z 243.196,A -85,B 0,C 180,E1 -16690.643,E2 -16690.643} C_VEL
LIN {X 0,Y 291.291,Z 243.2,A -85,B 0,C 180,E1 -16694.402,E2 -16694.402} C_VEL
LIN {X 0,Y 291.295,Z 243.2,A -85,B 0,C 180,E1 -16698.411,E2 -16698.411} C_VEL
LIN {X 0,Y 291.335,Z 243.195,A -85,B 0,C 180,E1 -16701.155,E2 -16701.155} C_VEL
LIN {X 0,Y 291.355,Z 243.19,A -85,B 0,C 180,E1 -16704.625,E2 -16704.625} C_VEL
LIN {X 0,Y 291.367,Z 243.191,A -85,B 0,C 180,E1 -16707.95,E2 -16707.95} C_VEL
LIN {X 0,Y 291.355,Z 243.185,A -85,B 0,C 180,E1 -16711.155,E2 -16711.155} C_VEL
LIN {X 0,Y 291.377,Z 243.18,A -85,B 0,C 180,E1 -16714.268,E2 -16714.268} C_VEL
LIN {X 0,Y 291.372,Z 243.19,A -85,B 0,C 180,E1 -16717.299,E2 -16717.299} C_VEL
LIN {X 0,Y 291.44,Z 243.18,A -85,B 0,C 180,E1 -16720.269,E2 -16720.269} C_VEL
LIN {X 0,Y 291.515,Z 243.168,A -85,B 0,C 180,E1 -16724.653,E2 -16724.653} C_VEL
LIN {X 0,Y 291.537,Z 243.161,A -85,B 0,C 180,E1 -16728.881,E2 -16728.881} C_VEL
LIN {X 0,Y 291.707,Z 243.143,A -85,B 0,C 180,E1 -16731.689,E2 -16731.689} C_VEL
LIN {X 0,Y 291.625,Z 243.154,A -85,B 0,C 180,E1 -16734.468,E2 -16734.468} C_VEL
LIN {X 0,Y 291.886,Z 243.116,A -85,B 0,C 180,E1 -16738.62,E2 -16738.62} C_VEL
LIN {X 0,Y 291.887,Z 243.124,A -85,B 0,C 180,E1 -16741.38,E2 -16741.38} C_VEL
LIN {X 0,Y 291.654,Z 243.152,A -85,B 0,C 180,E1 -16746.537,E2 -16746.537} C_VEL
LIN {X 0,Y 291.569,Z 243.163,A -85,B 0,C 180,E1 -16749.714,E2 -16749.714} C_VEL
LIN {X 0,Y 291.516,Z 243.164,A -85,B 0,C 180,E1 -16753.951,E2 -16753.951} C_VEL
LIN {X 0,Y 291.449,Z 243.169,A -85,B 0,C 180,E1 -16758.269,E2 -16758.269} C_VEL
LIN {X 0,Y 291.375,Z 243.186,A -85,B 0,C 180,E1 -16761.211,E2 -16761.211} C_VEL
LIN {X 0,Y 291.401,Z 243.184,A -85,B 0,C 180,E1 -16764.205,E2 -16764.205} C_VEL
LIN {X 0,Y 291.42,Z 243.178,A -85,B 0,C 180,E1 -16767.272,E2 -16767.272} C_VEL
LIN {X 0,Y 291.336,Z 243.189,A -85,B 0,C 180,E1 -16770.437,E2 -16770.437} C_VEL
LIN {X 0,Y 291.346,Z 243.19,A -85,B 0,C 180,E1 -16773.699,E2 -16773.699} C_VEL
LIN {X 0,Y 291.396,Z 243.186,A -85,B 0,C 180,E1 -16777.259,E2 -16777.259} C_VEL
LIN {X 0,Y 291.336,Z 243.195,A -85,B 0,C 180,E1 -16780.642,E2 -16780.642} C_VEL
LIN {X 0,Y 291.316,Z 243.199,A -85,B 0,C 180,E1 -16784.397,E2 -16784.397} C_VEL
LIN {X 0,Y 291.302,Z 243.205,A -85,B 0,C 180,E1 -16788.41,E2 -16788.41} C_VEL
LIN {X 0,Y 291.362,Z 243.206,A -85,B 0,C 180,E1 -16792.012,E2 -16792.012} C_VEL
LIN {X 0,Y 292.944,Z 249.453,A -85,B 0,C 180,E1 -16794.37,E2 -16794.37} C_VEL
LIN {X 0,Y 301.79,Z 267.767,A -85,B 0,C 180,E1 -16795.928,E2 -16795.928} C_VEL
LIN {X 0,Y 307.982,Z 282.582,A -85,B 0,C 180,E1 -16797.003,E2 -16797.003} C_VEL
LIN {X 0,Y 308.587,Z 286.235,A -85,B 0,C 180,E1 -16797.163,E2 -16797.163} C_VEL
LIN {X 0,Y 306.346,Z 357.067,A -85,B 0,C 180,E1 -16798.828,E2 -16798.828} C_VEL
LIN {X 0,Y 305.398,Z 371.019,A -85,B 0,C 180,E1 -16799.44,E2 -16799.44} C_VEL
LIN {X 0,Y 304.191,Z 382.938,A -85,B 0,C 180,E1 -16800.216,E2 -16800.216} C_VEL
LIN {X 0,Y 302.677,Z 394.173,A -85,B 0,C 180,E1 -16801.197,E2 -16801.197} C_VEL
LIN {X 0,Y 301.036,Z 404.957,A -85,B 0,C 180,E1 -16802.417,E2 -16802.417} C_VEL
LIN {X 0,Y 299.202,Z 415.206,A -85,B 0,C 180,E1 -16803.869,E2 -16803.869} C_VEL
LIN {X 0,Y 297.177,Z 424.801,A -85,B 0,C 180,E1 -16805.552,E2 -16805.552} C_VEL
LIN {X 0,Y 295.269,Z 433.997,A -85,B 0,C 180,E1 -16807.615,E2 -16807.615} C_VEL
LIN {X 0,Y 293.612,Z 441.373,A -85,B 0,C 180,E1 -16809.691,E2 -16809.691} C_VEL
LIN {X 0,Y 292.263,Z 447.262,A -85,B 0,C 180,E1 -16811.783,E2 -16811.783} C_VEL
LIN {X 0,Y 291.219,Z 451.882,A -85,B 0,C 180,E1 -16813.887,E2 -16813.887} C_VEL
LIN {X 0,Y 290.471,Z 455.381,A -85,B 0,C 180,E1 -16815.998,E2 -16815.998} C_VEL
LIN {X 0,Y 290.051,Z 457.133,A -85,B 0,C 180,E1 -16817.404,E2 -16817.404} C_VEL
LIN {X 0,Y 289.509,Z 459.383,A -85,B 0,C 180,E1 -16820.216,E2 -16820.216} C_VEL
LIN {X 0,Y 289.447,Z 459.916,A -85,B 0,C 180,E1 -16821.623,E2 -16821.623} C_VEL
LIN {X 0,Y 289.441,Z 460.015,A -85,B 0,C 180,E1 -16823.027,E2 -16823.027} C_VEL
LIN {X 0,Y 289.434,Z 459.664,A -85,B 0,C 180,E1 -16824.6,E2 -16824.6} C_VEL
LIN {X 0,Y 289.506,Z 457.996,A -85,B 0,C 180,E1 -16827.217,E2 -16827.217} C_VEL
LIN {X 0,Y 289.546,Z 456.494,A -85,B 0,C 180,E1 -16828.609,E2 -16828.609} C_VEL
LIN {X 0,Y 289.904,Z 453.464,A -85,B 0,C 180,E1 -16830.694,E2 -16830.694} C_VEL
LIN {X 0,Y 290.328,Z 449.398,A -85,B 0,C 180,E1 -16832.775,E2 -16832.775} C_VEL
LIN {X 0,Y 291.192,Z 443.167,A -85,B 0,C 180,E1 -16835.193,E2 -16835.193} C_VEL
LIN {X 0,Y 292.176,Z 436.392,A -85,B 0,C 180,E1 -16837.255,E2 -16837.255} C_VEL
LIN {X 0,Y 293.231,Z 429.479,A -85,B 0,C 180,E1 -16838.962,E2 -16838.962} C_VEL
LIN {X 0,Y 294.522,Z 421.156,A -85,B 0,C 180,E1 -16840.657,E2 -16840.657} C_VEL
LIN {X 0,Y 295.897,Z 410.913,A -85,B 0,C 180,E1 -16842.343,E2 -16842.343} C_VEL
LIN {X 0,Y 297.308,Z 399.426,A -85,B 0,C 180,E1 -16843.84,E2 -16843.84} C_VEL
LIN {X 0,Y 298.569,Z 387.931,A -85,B 0,C 180,E1 -16845.006,E2 -16845.006} C_VEL
LIN {X 0,Y 299.641,Z 375.489,A -85,B 0,C 180,E1 -16845.951,E2 -16845.951} C_VEL
LIN {X 0,Y 300.391,Z 362.419,A -85,B 0,C 180,E1 -16846.655,E2 -16846.655} C_VEL
LIN {X 0,Y 300.876,Z 349.947,A -85,B 0,C 180,E1 -16847.064,E2 -16847.064} C_VEL
LIN {X 0,Y 302.556,Z 281.028,A -85,B 0,C 180,E1 -16848.668,E2 -16848.668} C_VEL
LIN {X 0,Y 300.263,Z 269.045,A -85,B 0,C 180,E1 -16849.153,E2 -16849.153} C_VEL
LIN {X 0,Y 293.192,Z 250.488,A -85,B 0,C 180,E1 -16850.223,E2 -16850.223} C_VEL
LIN {X 0,Y 292.663,Z 248.873,A -85,B 0,C 180,E1 -16850.327,E2 -16850.327} C_VEL
LIN {X 0,Y 291.378,Z 243.191,A -85,B 0,C 180,E1 -16852.327,E2 -16852.327} C_VEL
LIN {X 0,Y 291.378,Z 243.189,A -85,B 0,C 180,E1 -16855.732,E2 -16855.732} C_VEL
LIN {X 0,Y 291.372,Z 243.189,A -85,B 0,C 180,E1 -16859.734,E2 -16859.734} C_VEL
LIN {X 0,Y 291.346,Z 243.191,A -85,B 0,C 180,E1 -16863.698,E2 -16863.698} C_VEL
LIN {X 0,Y 291.378,Z 243.188,A -85,B 0,C 180,E1 -16867.254,E2 -16867.254} C_VEL
LIN {X 0,Y 291.335,Z 243.197,A -85,B 0,C 180,E1 -16870.642,E2 -16870.642} C_VEL
LIN {X 0,Y 291.316,Z 243.197,A -85,B 0,C 180,E1 -16874.397,E2 -16874.397} C_VEL
LIN {X 0,Y 291.328,Z 243.196,A -85,B 0,C 180,E1 -16878.404,E2 -16878.404} C_VEL
LIN {X 0,Y 291.348,Z 243.191,A -85,B 0,C 180,E1 -16881.157,E2 -16881.157} C_VEL
LIN {X 0,Y 291.351,Z 243.191,A -85,B 0,C 180,E1 -16884.335,E2 -16884.335} C_VEL
LIN {X 0,Y 290.727,Z 243.275,A -85,B 0,C 180,E1 -16885.488,E2 -16885.488} C_VEL
LIN {X 0,Y 287.942,Z 243.626,A -85,B 0,C 180,E1 -16887.367,E2 -16887.367} C_VEL
LIN {X 0,Y 285.533,Z 243.922,A -85,B 0,C 180,E1 -16888.892,E2 -16888.892} C_VEL
LIN {X 0,Y 284.457,Z 244.049,A -85,B 0,C 180,E1 -16890.072,E2 -16890.072} C_VEL
LIN {X 0,Y 284.348,Z 244.06,A -85,B 0,C 180,E1 -16890.472,E2 -16890.472} C_VEL
LIN {X 0,Y 284.376,Z 244.058,A -85,B 0,C 180,E1 -16893.586,E2 -16893.586} C_VEL
LIN {X 0,Y 284.367,Z 244.05,A -85,B 0,C 180,E1 -16896.707,E2 -16896.707} C_VEL
LIN {X 0,Y 284.404,Z 244.054,A -85,B 0,C 180,E1 -16901.261,E2 -16901.261} C_VEL
LIN {X 0,Y 284.493,Z 244.047,A -85,B 0,C 180,E1 -16904.459,E2 -16904.459} C_VEL
LIN {X 0,Y 284.483,Z 244.032,A -85,B 0,C 180,E1 -16908.601,E2 -16908.601} C_VEL
LIN {X 0,Y 284.61,Z 244.024,A -85,B 0,C 180,E1 -16911.479,E2 -16911.479} C_VEL
LIN {X 0,Y 284.579,Z 244.035,A -85,B 0,C 180,E1 -16914.331,E2 -16914.331} C_VEL
LIN {X 0,Y 284.854,Z 243.999,A -85,B 0,C 180,E1 -16918.586,E2 -16918.586} C_VEL
LIN {X 0,Y 284.854,Z 243.999,A -85,B 0,C 180,E1 -16921.414,E2 -16921.414} C_VEL
LIN {X 0,Y 284.699,Z 244.02,A -85,B 0,C 180,E1 -16927.09,E2 -16927.09} C_VEL
LIN {X 0,Y 284.567,Z 244.033,A -85,B 0,C 180,E1 -16929.955,E2 -16929.955} C_VEL
LIN {X 0,Y 284.464,Z 244.05,A -85,B 0,C 180,E1 -16934.304,E2 -16934.304} C_VEL
LIN {X 0,Y 284.341,Z 244.062,A -85,B 0,C 180,E1 -16938.743,E2 -16938.743} C_VEL
LIN {X 0,Y 284.312,Z 244.067,A -85,B 0,C 180,E1 -16941.764,E2 -16941.764} C_VEL
LIN {X 0,Y 284.314,Z 244.066,A -85,B 0,C 180,E1 -16944.849,E2 -16944.849} C_VEL
LIN {X 0,Y 284.289,Z 244.072,A -85,B 0,C 180,E1 -16948.015,E2 -16948.015} C_VEL
LIN {X 0,Y 284.286,Z 244.07,A -85,B 0,C 180,E1 -16951.275,E2 -16951.275} C_VEL
LIN {X 0,Y 284.34,Z 244.063,A -85,B 0,C 180,E1 -16955.348,E2 -16955.348} C_VEL
LIN {X 0,Y 284.301,Z 244.071,A -85,B 0,C 180,E1 -16958.171,E2 -16958.171} C_VEL
LIN {X 0,Y 284.237,Z 244.078,A -85,B 0,C 180,E1 -16962.117,E2 -16962.117} C_VEL
LIN {X 0,Y 284.256,Z 244.076,A -85,B 0,C 180,E1 -16966.189,E2 -16966.189} C_VEL
LIN {X 0,Y 284.307,Z 244.068,A -85,B 0,C 180,E1 -16970.024,E2 -16970.024} C_VEL
LIN {X 0,Y 284.349,Z 244.065,A -85,B 0,C 180,E1 -16973.617,E2 -16973.617} C_VEL
LIN {X 0,Y 284.336,Z 244.113,A -85,B 0,C 180,E1 -16977.006,E2 -16977.006} C_VEL
LIN {X 0,Y 286.684,Z 254.888,A -85,B 0,C 180,E1 -16980.64,E2 -16980.64} C_VEL
LIN {X 0,Y 288.247,Z 263.206,A -85,B 0,C 180,E1 -16983.313,E2 -16983.313} C_VEL
LIN {X 0,Y 290.02,Z 269.375,A -85,B 0,C 180,E1 -16983.648,E2 -16983.648} C_VEL
LIN {X 0,Y 294.073,Z 296.365,A -85,B 0,C 180,E1 -16984.696,E2 -16984.696} C_VEL
LIN {X 0,Y 295.439,Z 307.483,A -85,B 0,C 180,E1 -16985.093,E2 -16985.093} C_VEL
LIN {X 0,Y 293.795,Z 371.868,A -85,B 0,C 180,E1 -16986.659,E2 -16986.659} C_VEL
LIN {X 0,Y 292.959,Z 385.087,A -85,B 0,C 180,E1 -16987.242,E2 -16987.242} C_VEL
LIN {X 0,Y 291.841,Z 397.805,A -85,B 0,C 180,E1 -16988.083,E2 -16988.083} C_VEL
LIN {X 0,Y 290.54,Z 409.083,A -85,B 0,C 180,E1 -16989.097,E2 -16989.097} C_VEL
LIN {X 0,Y 288.978,Z 420.76,A -85,B 0,C 180,E1 -16990.464,E2 -16990.464} C_VEL
LIN {X 0,Y 287.484,Z 431.269,A -85,B 0,C 180,E1 -16992.023,E2 -16992.023} C_VEL
LIN {X 0,Y 286.358,Z 440.099,A -85,B 0,C 180,E1 -16993.655,E2 -16993.655} C_VEL
LIN {X 0,Y 285.209,Z 447.768,A -85,B 0,C 180,E1 -16995.37,E2 -16995.37} C_VEL
LIN {X 0,Y 283.97,Z 455.47,A -85,B 0,C 180,E1 -16997.493,E2 -16997.493} C_VEL
LIN {X 0,Y 283.124,Z 462.579,A -85,B 0,C 180,E1 -16999.993,E2 -16999.993} C_VEL
LIN {X 0,Y 282.669,Z 467.294,A -85,B 0,C 180,E1 -17002.14,E2 -17002.14} C_VEL
LIN {X 0,Y 282.371,Z 471.343,A -85,B 0,C 180,E1 -17004.607,E2 -17004.607} C_VEL
LIN {X 0,Y 282.347,Z 474.098,A -85,B 0,C 180,E1 -17007.147,E2 -17007.147} C_VEL
LIN {X 0,Y 282.339,Z 475.074,A -85,B 0,C 180,E1 -17008.574,E2 -17008.574} C_VEL
LIN {X 0,Y 282.355,Z 475.659,A -85,B 0,C 180,E1 -17010,E2 -17010} C_VEL
LIN {X 0,Y 282.33,Z 475.838,A -85,B 0,C 180,E1 -17011.426,E2 -17011.426} C_VEL
LIN {X 0,Y 282.336,Z 475.59,A -85,B 0,C 180,E1 -17012.854,E2 -17012.854} C_VEL
LIN {X 0,Y 282.388,Z 473.937,A -85,B 0,C 180,E1 -17015.713,E2 -17015.713} C_VEL
LIN {X 0,Y 282.578,Z 472.514,A -85,B 0,C 180,E1 -17017.144,E2 -17017.144} C_VEL
LIN {X 0,Y 283.054,Z 469.555,A -85,B 0,C 180,E1 -17019.288,E2 -17019.288} C_VEL
LIN {X 0,Y 283.833,Z 465.567,A -85,B 0,C 180,E1 -17021.425,E2 -17021.425} C_VEL
LIN {X 0,Y 285.123,Z 459.454,A -85,B 0,C 180,E1 -17023.906,E2 -17023.906} C_VEL
LIN {X 0,Y 286.798,Z 452.797,A -85,B 0,C 180,E1 -17026.003,E2 -17026.003} C_VEL
LIN {X 0,Y 288.562,Z 444.762,A -85,B 0,C 180,E1 -17028.039,E2 -17028.039} C_VEL
LIN {X 0,Y 290.299,Z 436.122,A -85,B 0,C 180,E1 -17029.812,E2 -17029.812} C_VEL
LIN {X 0,Y 292.522,Z 425.717,A -85,B 0,C 180,E1 -17031.493,E2 -17031.493} C_VEL
LIN {X 0,Y 294.644,Z 414.021,A -85,B 0,C 180,E1 -17032.991,E2 -17032.991} C_VEL
LIN {X 0,Y 296.558,Z 402.332,A -85,B 0,C 180,E1 -17034.13,E2 -17034.13} C_VEL
LIN {X 0,Y 298.105,Z 390.199,A -85,B 0,C 180,E1 -17035.017,E2 -17035.017} C_VEL
LIN {X 0,Y 299.356,Z 376.968,A -85,B 0,C 180,E1 -17035.696,E2 -17035.696} C_VEL
LIN {X 0,Y 300.066,Z 363.948,A -85,B 0,C 180,E1 -17036.097,E2 -17036.097} C_VEL
LIN {X 0,Y 301.599,Z 308.916,A -85,B 0,C 180,E1 -17037.408,E2 -17037.408} C_VEL
LIN {X 0,Y 297.02,Z 283.124,A -85,B 0,C 180,E1 -17038.624,E2 -17038.624} C_VEL
LIN {X 0,Y 295.929,Z 278.961,A -85,B 0,C 180,E1 -17038.867,E2 -17038.867} C_VEL
LIN {X 0,Y 288.82,Z 262.716,A -85,B 0,C 180,E1 -17040.218,E2 -17040.218} C_VEL
LIN {X 0,Y 286.494,Z 252.758,A -85,B 0,C 180,E1 -17043.81,E2 -17043.81} C_VEL
LIN {X 0,Y 284.363,Z 244.064,A -85,B 0,C 180,E1 -17047.155,E2 -17047.155} C_VEL
LIN {X 0,Y 284.306,Z 244.073,A -85,B 0,C 180,E1 -17049.995,E2 -17049.995} C_VEL
LIN {X 0,Y 284.246,Z 244.078,A -85,B 0,C 180,E1 -17054.19,E2 -17054.19} C_VEL
LIN {X 0,Y 284.241,Z 244.079,A -85,B 0,C 180,E1 -17058.119,E2 -17058.119} C_VEL
LIN {X 0,Y 284.309,Z 244.066,A -85,B 0,C 180,E1 -17062.282,E2 -17062.282} C_VEL
LIN {X 0,Y 284.307,Z 244.069,A -85,B 0,C 180,E1 -17065.351,E2 -17065.351} C_VEL
LIN {X 0,Y 284.287,Z 244.072,A -85,B 0,C 180,E1 -17068.725,E2 -17068.725} C_VEL
LIN {X 0,Y 284.292,Z 244.072,A -85,B 0,C 180,E1 -17071.985,E2 -17071.985} C_VEL
LIN {X 0,Y 284.326,Z 244.068,A -85,B 0,C 180,E1 -17076.145,E2 -17076.145} C_VEL
LIN {X 0,Y 284.377,Z 244.059,A -85,B 0,C 180,E1 -17079.904,E2 -17079.904} C_VEL
LIN {X 0,Y 284.455,Z 244.048,A -85,B 0,C 180,E1 -17084.487,E2 -17084.487} C_VEL
LIN {X 0,Y 284.489,Z 244.038,A -85,B 0,C 180,E1 -17088.602,E2 -17088.602} C_VEL
LIN {X 0,Y 284.658,Z 244.022,A -85,B 0,C 180,E1 -17091.481,E2 -17091.481} C_VEL
LIN {X 0,Y 284.596,Z 244.03,A -85,B 0,C 180,E1 -17094.331,E2 -17094.331} C_VEL
LIN {X 0,Y 284.852,Z 243.992,A -85,B 0,C 180,E1 -17098.586,E2 -17098.586} C_VEL
LIN {X 0,Y 284.854,Z 244,A -85,B 0,C 180,E1 -17101.414,E2 -17101.414} C_VEL
LIN {X 0,Y 284.649,Z 244.023,A -85,B 0,C 180,E1 -17107.091,E2 -17107.091} C_VEL
LIN {X 0,Y 284.515,Z 244.044,A -85,B 0,C 180,E1 -17109.957,E2 -17109.957} C_VEL
LIN {X 0,Y 284.464,Z 244.045,A -85,B 0,C 180,E1 -17114.304,E2 -17114.304} C_VEL
LIN {X 0,Y 284.387,Z 244.05,A -85,B 0,C 180,E1 -17118.74,E2 -17118.74} C_VEL
LIN {X 0,Y 284.368,Z 244.054,A -85,B 0,C 180,E1 -17123.293,E2 -17123.293} C_VEL
LIN {X 0,Y 284.396,Z 244.052,A -85,B 0,C 180,E1 -17127.173,E2 -17127.173} C_VEL
LIN {X 0,Y 284.295,Z 244.07,A -85,B 0,C 180,E1 -17131.275,E2 -17131.275} C_VEL
LIN {X 0,Y 284.363,Z 244.064,A -85,B 0,C 180,E1 -17135.354,E2 -17135.354} C_VEL
LIN {X 0,Y 284.325,Z 244.067,A -85,B 0,C 180,E1 -17138.167,E2 -17138.167} C_VEL
LIN {X 0,Y 284.271,Z 244.075,A -85,B 0,C 180,E1 -17142.125,E2 -17142.125} C_VEL
LIN {X 0,Y 284.27,Z 244.068,A -85,B 0,C 180,E1 -17146.192,E2 -17146.192} C_VEL
LIN {X 0,Y 284.285,Z 244.071,A -85,B 0,C 180,E1 -17150.03,E2 -17150.03} C_VEL
LIN {X 0,Y 284.314,Z 244.086,A -85,B 0,C 180,E1 -17151.266,E2 -17151.266} C_VEL
LIN {X 0,Y 285.731,Z 249.593,A -85,B 0,C 180,E1 -17153.45,E2 -17153.45} C_VEL
LIN {X 0,Y 294.969,Z 268.372,A -85,B 0,C 180,E1 -17155.151,E2 -17155.151} C_VEL
LIN {X 0,Y 301.999,Z 284.846,A -85,B 0,C 180,E1 -17156.414,E2 -17156.414} C_VEL
LIN {X 0,Y 302.385,Z 287.794,A -85,B 0,C 180,E1 -17156.536,E2 -17156.536} C_VEL
LIN {X 0,Y 300.085,Z 357.317,A -85,B 0,C 180,E1 -17158.2,E2 -17158.2} C_VEL
LIN {X 0,Y 299.103,Z 371.252,A -85,B 0,C 180,E1 -17158.824,E2 -17158.824} C_VEL
LIN {X 0,Y 297.846,Z 383.16,A -85,B 0,C 180,E1 -17159.613,E2 -17159.613} C_VEL
LIN {X 0,Y 296.148,Z 395.187,A -85,B 0,C 180,E1 -17160.695,E2 -17160.695} C_VEL
LIN {X 0,Y 294.298,Z 406.568,A -85,B 0,C 180,E1 -17162.035,E2 -17162.035} C_VEL
LIN {X 0,Y 292.315,Z 417.016,A -85,B 0,C 180,E1 -17163.59,E2 -17163.59} C_VEL
LIN {X 0,Y 290.624,Z 424.562,A -85,B 0,C 180,E1 -17164.964,E2 -17164.964} C_VEL
LIN {X 0,Y 288.942,Z 432.479,A -85,B 0,C 180,E1 -17166.718,E2 -17166.718} C_VEL
LIN {X 0,Y 287.103,Z 440.171,A -85,B 0,C 180,E1 -17168.834,E2 -17168.834} C_VEL
LIN {X 0,Y 285.413,Z 447.235,A -85,B 0,C 180,E1 -17171.33,E2 -17171.33} C_VEL
LIN {X 0,Y 284.304,Z 451.903,A -85,B 0,C 180,E1 -17173.484,E2 -17173.484} C_VEL
LIN {X 0,Y 283.488,Z 455.445,A -85,B 0,C 180,E1 -17175.646,E2 -17175.646} C_VEL
LIN {X 0,Y 283.046,Z 457.241,A -85,B 0,C 180,E1 -17177.087,E2 -17177.087} C_VEL
LIN {X 0,Y 282.459,Z 459.531,A -85,B 0,C 180,E1 -17179.97,E2 -17179.97} C_VEL
LIN {X 0,Y 282.355,Z 460.089,A -85,B 0,C 180,E1 -17181.411,E2 -17181.411} C_VEL
LIN {X 0,Y 282.336,Z 460.223,A -85,B 0,C 180,E1 -17182.85,E2 -17182.85} C_VEL
LIN {X 0,Y 282.349,Z 459.825,A -85,B 0,C 180,E1 -17184.656,E2 -17184.656} C_VEL
LIN {X 0,Y 282.429,Z 458.265,A -85,B 0,C 180,E1 -17187.147,E2 -17187.147} C_VEL
LIN {X 0,Y 282.462,Z 456.801,A -85,B 0,C 180,E1 -17188.574,E2 -17188.574} C_VEL
LIN {X 0,Y 282.803,Z 453.814,A -85,B 0,C 180,E1 -17190.712,E2 -17190.712} C_VEL
LIN {X 0,Y 283.247,Z 449.793,A -85,B 0,C 180,E1 -17192.844,E2 -17192.844} C_VEL
LIN {X 0,Y 284.16,Z 443.611,A -85,B 0,C 180,E1 -17195.322,E2 -17195.322} C_VEL
LIN {X 0,Y 285.16,Z 436.892,A -85,B 0,C 180,E1 -17197.434,E2 -17197.434} C_VEL
LIN {X 0,Y 286.549,Z 428.534,A -85,B 0,C 180,E1 -17199.529,E2 -17199.529} C_VEL
LIN {X 0,Y 287.769,Z 419.941,A -85,B 0,C 180,E1 -17201.267,E2 -17201.267} C_VEL
LIN {X 0,Y 289.332,Z 409.352,A -85,B 0,C 180,E1 -17202.984,E2 -17202.984} C_VEL
LIN {X 0,Y 290.774,Z 397.92,A -85,B 0,C 180,E1 -17204.455,E2 -17204.455} C_VEL
LIN {X 0,Y 292.021,Z 386.368,A -85,B 0,C 180,E1 -17205.599,E2 -17205.599} C_VEL
LIN {X 0,Y 293.114,Z 373.58,A -85,B 0,C 180,E1 -17206.55,E2 -17206.55} C_VEL
LIN {X 0,Y 293.823,Z 360.602,A -85,B 0,C 180,E1 -17207.217,E2 -17207.217} C_VEL
LIN {X 0,Y 294.367,Z 344.775,A -85,B 0,C 180,E1 -17207.678,E2 -17207.678} C_VEL
LIN {X 0,Y 295.918,Z 281.604,A -85,B 0,C 180,E1 -17209.183,E2 -17209.183} C_VEL
LIN {X 0,Y 294.049,Z 271.545,A -85,B 0,C 180,E1 -17209.599,E2 -17209.599} C_VEL
LIN {X 0,Y 286.64,Z 252.022,A -85,B 0,C 180,E1 -17210.763,E2 -17210.763} C_VEL
LIN {X 0,Y 285.431,Z 248.992,A -85,B 0,C 180,E1 -17210.999,E2 -17210.999} C_VEL
LIN {X 0,Y 284.332,Z 244.069,A -85,B 0,C 180,E1 -17212.815,E2 -17212.815} C_VEL
LIN {X 0,Y 284.346,Z 244.066,A -85,B 0,C 180,E1 -17217.152,E2 -17217.152} C_VEL
LIN {X 0,Y 284.302,Z 244.07,A -85,B 0,C 180,E1 -17220.093,E2 -17220.093} C_VEL
LIN {X 0,Y 284.306,Z 244.071,A -85,B 0,C 180,E1 -17222.945,E2 -17222.945} C_VEL
LIN {X 0,Y 284.334,Z 244.067,A -85,B 0,C 180,E1 -17226.386,E2 -17226.386} C_VEL
LIN {X 0,Y 284.307,Z 244.068,A -85,B 0,C 180,E1 -17229.994,E2 -17229.994} C_VEL
LIN {X 0,Y 284.267,Z 244.074,A -85,B 0,C 180,E1 -17234.194,E2 -17234.194} C_VEL
LIN {X 0,Y 284.273,Z 244.073,A -85,B 0,C 180,E1 -17238.124,E2 -17238.124} C_VEL
LIN {X 0,Y 284.32,Z 244.067,A -85,B 0,C 180,E1 -17242.279,E2 -17242.279} C_VEL
LIN {X 0,Y 284.309,Z 244.065,A -85,B 0,C 180,E1 -17245.351,E2 -17245.351} C_VEL
LIN {X 0,Y 284.295,Z 244.063,A -85,B 0,C 180,E1 -17248.725,E2 -17248.725} C_VEL
LIN {X 0,Y 284.348,Z 244.06,A -85,B 0,C 180,E1 -17250.472,E2 -17250.472} C_VEL
LIN {X 0,Y 283.631,Z 244.152,A -85,B 0,C 180,E1 -17251.655,E2 -17251.655} C_VEL
LIN {X 0,Y 280.793,Z 244.505,A -85,B 0,C 180,E1 -17253.583,E2 -17253.583} C_VEL
LIN {X 0,Y 278.41,Z 244.799,A -85,B 0,C 180,E1 -17255.148,E2 -17255.148} C_VEL
LIN {X 0,Y 277.377,Z 244.923,A -85,B 0,C 180,E1 -17256.36,E2 -17256.36} C_VEL
LIN {X 0,Y 277.285,Z 244.929,A -85,B 0,C 180,E1 -17256.77,E2 -17256.77} C_VEL
LIN {X 0,Y 277.346,Z 244.934,A -85,B 0,C 180,E1 -17260.766,E2 -17260.766} C_VEL
LIN {X 0,Y 277.436,Z 244.919,A -85,B 0,C 180,E1 -17265.326,E2 -17265.326} C_VEL
LIN {X 0,Y 277.458,Z 244.906,A -85,B 0,C 180,E1 -17269.787,E2 -17269.787} C_VEL
LIN {X 0,Y 277.604,Z 244.903,A -85,B 0,C 180,E1 -17272.728,E2 -17272.728} C_VEL
LIN {X 0,Y 277.82,Z 244.875,A -85,B 0,C 180,E1 -17278.55,E2 -17278.55} C_VEL
LIN {X 0,Y 277.82,Z 244.875,A -85,B 0,C 180,E1 -17281.449,E2 -17281.449} C_VEL
LIN {X 0,Y 277.654,Z 244.897,A -85,B 0,C 180,E1 -17287.271,E2 -17287.271} C_VEL
LIN {X 0,Y 277.507,Z 244.914,A -85,B 0,C 180,E1 -17290.211,E2 -17290.211} C_VEL
LIN {X 0,Y 277.41,Z 244.931,A -85,B 0,C 180,E1 -17294.675,E2 -17294.675} C_VEL
LIN {X 0,Y 277.304,Z 244.937,A -85,B 0,C 180,E1 -17299.237,E2 -17299.237} C_VEL
LIN {X 0,Y 277.286,Z 244.942,A -85,B 0,C 180,E1 -17303.924,E2 -17303.924} C_VEL
LIN {X 0,Y 277.274,Z 244.944,A -85,B 0,C 180,E1 -17307.485,E2 -17307.485} C_VEL
LIN {X 0,Y 277.248,Z 244.947,A -85,B 0,C 180,E1 -17310.473,E2 -17310.473} C_VEL
LIN {X 0,Y 277.246,Z 244.948,A -85,B 0,C 180,E1 -17313.896,E2 -17313.896} C_VEL
LIN {X 0,Y 277.261,Z 244.946,A -85,B 0,C 180,E1 -17317.47,E2 -17317.47} C_VEL
LIN {X 0,Y 277.184,Z 244.956,A -85,B 0,C 180,E1 -17321.241,E2 -17321.241} C_VEL
LIN {X 0,Y 277.201,Z 244.953,A -85,B 0,C 180,E1 -17325.227,E2 -17325.227} C_VEL
LIN {X 0,Y 277.223,Z 244.949,A -85,B 0,C 180,E1 -17329.512,E2 -17329.512} C_VEL
LIN {X 0,Y 277.278,Z 244.948,A -85,B 0,C 180,E1 -17332.532,E2 -17332.532} C_VEL
LIN {X 0,Y 277.294,Z 244.946,A -85,B 0,C 180,E1 -17336.454,E2 -17336.454} C_VEL
LIN {X 0,Y 279.916,Z 257.042,A -85,B 0,C 180,E1 -17340.687,E2 -17340.687} C_VEL
LIN {X 0,Y 281.033,Z 262.97,A -85,B 0,C 180,E1 -17342.645,E2 -17342.645} C_VEL
LIN {X 0,Y 283.641,Z 270.973,A -85,B 0,C 180,E1 -17343.126,E2 -17343.126} C_VEL
LIN {X 0,Y 288.126,Z 301.478,A -85,B 0,C 180,E1 -17344.338,E2 -17344.338} C_VEL
LIN {X 0,Y 288.872,Z 308.534,A -85,B 0,C 180,E1 -17344.588,E2 -17344.588} C_VEL
LIN {X 0,Y 287.202,Z 371.202,A -85,B 0,C 180,E1 -17346.138,E2 -17346.138} C_VEL
LIN {X 0,Y 286.334,Z 384.578,A -85,B 0,C 180,E1 -17346.733,E2 -17346.733} C_VEL
LIN {X 0,Y 285.202,Z 396.804,A -85,B 0,C 180,E1 -17347.545,E2 -17347.545} C_VEL
LIN {X 0,Y 283.898,Z 408.312,A -85,B 0,C 180,E1 -17348.584,E2 -17348.584} C_VEL
LIN {X 0,Y 282.283,Z 420.108,A -85,B 0,C 180,E1 -17349.981,E2 -17349.981} C_VEL
LIN {X 0,Y 280.691,Z 430.69,A -85,B 0,C 180,E1 -17351.572,E2 -17351.572} C_VEL
LIN {X 0,Y 279.449,Z 440.02,A -85,B 0,C 180,E1 -17353.33,E2 -17353.33} C_VEL
LIN {X 0,Y 278.078,Z 448.713,A -85,B 0,C 180,E1 -17355.361,E2 -17355.361} C_VEL
LIN {X 0,Y 276.84,Z 456.205,A -85,B 0,C 180,E1 -17357.538,E2 -17357.538} C_VEL
LIN {X 0,Y 276.112,Z 462.225,A -85,B 0,C 180,E1 -17359.737,E2 -17359.737} C_VEL
LIN {X 0,Y 275.595,Z 466.973,A -85,B 0,C 180,E1 -17361.937,E2 -17361.937} C_VEL
LIN {X 0,Y 275.337,Z 470.596,A -85,B 0,C 180,E1 -17364.14,E2 -17364.14} C_VEL
LIN {X 0,Y 275.25,Z 472.459,A -85,B 0,C 180,E1 -17365.607,E2 -17365.607} C_VEL
LIN {X 0,Y 275.256,Z 473.853,A -85,B 0,C 180,E1 -17367.073,E2 -17367.073} C_VEL
LIN {X 0,Y 275.263,Z 474.844,A -85,B 0,C 180,E1 -17368.537,E2 -17368.537} C_VEL
LIN {X 0,Y 275.277,Z 475.442,A -85,B 0,C 180,E1 -17370,E2 -17370} C_VEL
LIN {X 0,Y 275.255,Z 475.645,A -85,B 0,C 180,E1 -17371.463,E2 -17371.463} C_VEL
LIN {X 0,Y 275.245,Z 475.414,A -85,B 0,C 180,E1 -17372.927,E2 -17372.927} C_VEL
LIN {X 0,Y 275.302,Z 473.788,A -85,B 0,C 180,E1 -17375.861,E2 -17375.861} C_VEL
LIN {X 0,Y 275.512,Z 472.387,A -85,B 0,C 180,E1 -17377.328,E2 -17377.328} C_VEL
LIN {X 0,Y 276.016,Z 469.452,A -85,B 0,C 180,E1 -17379.527,E2 -17379.527} C_VEL
LIN {X 0,Y 276.842,Z 465.495,A -85,B 0,C 180,E1 -17381.718,E2 -17381.718} C_VEL
LIN {X 0,Y 277.97,Z 460.418,A -85,B 0,C 180,E1 -17383.898,E2 -17383.898} C_VEL
LIN {X 0,Y 279.632,Z 454.047,A -85,B 0,C 180,E1 -17386.049,E2 -17386.049} C_VEL
LIN {X 0,Y 281.245,Z 447.225,A -85,B 0,C 180,E1 -17387.916,E2 -17387.916} C_VEL
LIN {X 0,Y 283.232,Z 438.024,A -85,B 0,C 180,E1 -17389.949,E2 -17389.949} C_VEL
LIN {X 0,Y 285.448,Z 428.183,A -85,B 0,C 180,E1 -17391.673,E2 -17391.673} C_VEL
LIN {X 0,Y 287.657,Z 417.165,A -85,B 0,C 180,E1 -17393.201,E2 -17393.201} C_VEL
LIN {X 0,Y 289.543,Z 406.38,A -85,B 0,C 180,E1 -17394.371,E2 -17394.371} C_VEL
LIN {X 0,Y 291.413,Z 393.38,A -85,B 0,C 180,E1 -17395.441,E2 -17395.441} C_VEL
LIN {X 0,Y 292.717,Z 380.791,A -85,B 0,C 180,E1 -17396.179,E2 -17396.179} C_VEL
LIN {X 0,Y 293.685,Z 367.582,A -85,B 0,C 180,E1 -17396.66,E2 -17396.66} C_VEL
LIN {X 0,Y 295.437,Z 309.967,A -85,B 0,C 180,E1 -17398.064,E2 -17398.064} C_VEL
LIN {X 0,Y 290.775,Z 283.522,A -85,B 0,C 180,E1 -17399.354,E2 -17399.354} C_VEL
LIN {X 0,Y 285.074,Z 270.173,A -85,B 0,C 180,E1 -17400.456,E2 -17400.456} C_VEL
LIN {X 0,Y 281.531,Z 262.546,A -85,B 0,C 180,E1 -17401.155,E2 -17401.155} C_VEL
LIN {X 0,Y 279.204,Z 252.344,A -85,B 0,C 180,E1 -17404.977,E2 -17404.977} C_VEL
LIN {X 0,Y 277.272,Z 244.948,A -85,B 0,C 180,E1 -17407.961,E2 -17407.961} C_VEL
LIN {X 0,Y 277.21,Z 244.956,A -85,B 0,C 180,E1 -17411.236,E2 -17411.236} C_VEL
LIN {X 0,Y 277.201,Z 244.957,A -85,B 0,C 180,E1 -17415.226,E2 -17415.226} C_VEL
LIN {X 0,Y 277.197,Z 244.957,A -85,B 0,C 180,E1 -17419.518,E2 -17419.518} C_VEL
LIN {X 0,Y 277.255,Z 244.944,A -85,B 0,C 180,E1 -17422.529,E2 -17422.529} C_VEL
LIN {X 0,Y 277.246,Z 244.942,A -85,B 0,C 180,E1 -17426.104,E2 -17426.104} C_VEL
LIN {X 0,Y 277.262,Z 244.942,A -85,B 0,C 180,E1 -17429.539,E2 -17429.539} C_VEL
LIN {X 0,Y 277.306,Z 244.942,A -85,B 0,C 180,E1 -17432.859,E2 -17432.859} C_VEL
LIN {X 0,Y 277.288,Z 244.945,A -85,B 0,C 180,E1 -17436.076,E2 -17436.076} C_VEL
LIN {X 0,Y 277.325,Z 244.939,A -85,B 0,C 180,E1 -17440.765,E2 -17440.765} C_VEL
LIN {X 0,Y 277.415,Z 244.929,A -85,B 0,C 180,E1 -17445.325,E2 -17445.325} C_VEL
LIN {X 0,Y 277.508,Z 244.917,A -85,B 0,C 180,E1 -17449.789,E2 -17449.789} C_VEL
LIN {X 0,Y 277.651,Z 244.888,A -85,B 0,C 180,E1 -17452.729,E2 -17452.729} C_VEL
LIN {X 0,Y 277.818,Z 244.867,A -85,B 0,C 180,E1 -17458.551,E2 -17458.551} C_VEL
LIN {X 0,Y 277.82,Z 244.875,A -85,B 0,C 180,E1 -17461.45,E2 -17461.45} C_VEL
LIN {X 0,Y 277.607,Z 244.898,A -85,B 0,C 180,E1 -17467.272,E2 -17467.272} C_VEL
LIN {X 0,Y 277.458,Z 244.922,A -85,B 0,C 180,E1 -17470.213,E2 -17470.213} C_VEL
LIN {X 0,Y 277.411,Z 244.924,A -85,B 0,C 180,E1 -17474.676,E2 -17474.676} C_VEL
LIN {X 0,Y 277.336,Z 244.931,A -85,B 0,C 180,E1 -17479.235,E2 -17479.235} C_VEL
LIN {X 0,Y 277.32,Z 244.938,A -85,B 0,C 180,E1 -17484.17,E2 -17484.17} C_VEL
LIN {X 0,Y 277.324,Z 244.936,A -85,B 0,C 180,E1 -17487.504,E2 -17487.504} C_VEL
LIN {X 0,Y 277.273,Z 244.94,A -85,B 0,C 180,E1 -17490.482,E2 -17490.482} C_VEL
LIN {X 0,Y 277.256,Z 244.946,A -85,B 0,C 180,E1 -17493.895,E2 -17493.895} C_VEL
LIN {X 0,Y 277.283,Z 244.946,A -85,B 0,C 180,E1 -17497.467,E2 -17497.467} C_VEL
LIN {X 0,Y 277.211,Z 244.952,A -85,B 0,C 180,E1 -17501.237,E2 -17501.237} C_VEL
LIN {X 0,Y 277.218,Z 244.955,A -85,B 0,C 180,E1 -17505.223,E2 -17505.223} C_VEL
LIN {X 0,Y 277.201,Z 244.955,A -85,B 0,C 180,E1 -17509.518,E2 -17509.518} C_VEL
LIN {X 0,Y 277.276,Z 245.075,A -85,B 0,C 180,E1 -17510.517,E2 -17510.517} C_VEL
LIN {X 0,Y 278.579,Z 249.966,A -85,B 0,C 180,E1 -17512.489,E2 -17512.489} C_VEL
LIN {X 0,Y 287.73,Z 267.95,A -85,B 0,C 180,E1 -17514.247,E2 -17514.247} C_VEL
LIN {X 0,Y 295.259,Z 285.228,A -85,B 0,C 180,E1 -17515.656,E2 -17515.656} C_VEL
LIN {X 0,Y 296.22,Z 287.692,A -85,B 0,C 180,E1 -17515.836,E2 -17515.836} C_VEL
LIN {X 0,Y 293.868,Z 357.501,A -85,B 0,C 180,E1 -17517.544,E2 -17517.544} C_VEL
LIN {X 0,Y 292.837,Z 371.484,A -85,B 0,C 180,E1 -17518.181,E2 -17518.181} C_VEL
LIN {X 0,Y 291.418,Z 384.411,A -85,B 0,C 180,E1 -17519.07,E2 -17519.07} C_VEL
LIN {X 0,Y 289.639,Z 396.201,A -85,B 0,C 180,E1 -17520.17,E2 -17520.17} C_VEL
LIN {X 0,Y 287.614,Z 407.95,A -85,B 0,C 180,E1 -17521.605,E2 -17521.605} C_VEL
LIN {X 0,Y 285.419,Z 418.704,A -85,B 0,C 180,E1 -17523.296,E2 -17523.296} C_VEL
LIN {X 0,Y 283.384,Z 427.691,A -85,B 0,C 180,E1 -17525.064,E2 -17525.064} C_VEL
LIN {X 0,Y 281.343,Z 436.435,A -85,B 0,C 180,E1 -17527.221,E2 -17527.221} C_VEL
LIN {X 0,Y 279.584,Z 443.372,A -85,B 0,C 180,E1 -17529.395,E2 -17529.395} C_VEL
LIN {X 0,Y 278.143,Z 448.908,A -85,B 0,C 180,E1 -17531.588,E2 -17531.588} C_VEL
LIN {X 0,Y 277.095,Z 453.232,A -85,B 0,C 180,E1 -17533.8,E2 -17533.8} C_VEL
LIN {X 0,Y 276.52,Z 455.513,A -85,B 0,C 180,E1 -17535.276,E2 -17535.276} C_VEL
LIN {X 0,Y 276.034,Z 457.348,A -85,B 0,C 180,E1 -17536.753,E2 -17536.753} C_VEL
LIN {X 0,Y 275.402,Z 459.679,A -85,B 0,C 180,E1 -17539.71,E2 -17539.71} C_VEL
LIN {X 0,Y 275.284,Z 460.257,A -85,B 0,C 180,E1 -17541.189,E2 -17541.189} C_VEL
LIN {X 0,Y 275.244,Z 460.43,A -85,B 0,C 180,E1 -17542.665,E2 -17542.665} C_VEL
LIN {X 0,Y 275.256,Z 459.98,A -85,B 0,C 180,E1 -17544.734,E2 -17544.734} C_VEL
LIN {X 0,Y 275.33,Z 458.531,A -85,B 0,C 180,E1 -17547.074,E2 -17547.074} C_VEL
LIN {X 0,Y 275.38,Z 457.106,A -85,B 0,C 180,E1 -17548.538,E2 -17548.538} C_VEL
LIN {X 0,Y 275.702,Z 454.158,A -85,B 0,C 180,E1 -17550.73,E2 -17550.73} C_VEL
LIN {X 0,Y 276.166,Z 450.18,A -85,B 0,C 180,E1 -17552.917,E2 -17552.917} C_VEL
LIN {X 0,Y 277.131,Z 444.051,A -85,B 0,C 180,E1 -17555.457,E2 -17555.457} C_VEL
LIN {X 0,Y 278.133,Z 437.388,A -85,B 0,C 180,E1 -17557.623,E2 -17557.623} C_VEL
LIN {X 0,Y 279.583,Z 429.111,A -85,B 0,C 180,E1 -17559.769,E2 -17559.769} C_VEL
LIN {X 0,Y 280.841,Z 420.61,A -85,B 0,C 180,E1 -17561.549,E2 -17561.549} C_VEL
LIN {X 0,Y 282.444,Z 410.118,A -85,B 0,C 180,E1 -17563.307,E2 -17563.307} C_VEL
LIN {X 0,Y 283.916,Z 399.102,A -85,B 0,C 180,E1 -17564.778,E2 -17564.778} C_VEL
LIN {X 0,Y 285.279,Z 387.182,A -85,B 0,C 180,E1 -17566.01,E2 -17566.01} C_VEL
LIN {X 0,Y 286.447,Z 373.956,A -85,B 0,C 180,E1 -17567.023,E2 -17567.023} C_VEL
LIN {X 0,Y 287.164,Z 361.816,A -85,B 0,C 180,E1 -17567.676,E2 -17567.676} C_VEL
LIN {X 0,Y 287.737,Z 348.395,A -85,B 0,C 180,E1 -17568.099,E2 -17568.099} C_VEL
LIN {X 0,Y 289.383,Z 282.564,A -85,B 0,C 180,E1 -17569.704,E2 -17569.704} C_VEL
LIN {X 0,Y 287.694,Z 273.712,A -85,B 0,C 180,E1 -17570.086,E2 -17570.086} C_VEL
LIN {X 0,Y 281.416,Z 257.007,A -85,B 0,C 180,E1 -17571.108,E2 -17571.108} C_VEL
LIN {X 0,Y 278.271,Z 249.229,A -85,B 0,C 180,E1 -17571.661,E2 -17571.661} C_VEL
LIN {X 0,Y 277.289,Z 244.945,A -85,B 0,C 180,E1 -17573.231,E2 -17573.231} C_VEL
LIN {X 0,Y 277.283,Z 244.944,A -85,B 0,C 180,E1 -17577.487,E2 -17577.487} C_VEL
LIN {X 0,Y 277.249,Z 244.951,A -85,B 0,C 180,E1 -17580.472,E2 -17580.472} C_VEL
LIN {X 0,Y 277.248,Z 244.948,A -85,B 0,C 180,E1 -17583.895,E2 -17583.895} C_VEL
LIN {X 0,Y 277.269,Z 244.945,A -85,B 0,C 180,E1 -17587.469,E2 -17587.469} C_VEL
LIN {X 0,Y 277.211,Z 244.952,A -85,B 0,C 180,E1 -17591.236,E2 -17591.236} C_VEL
LIN {X 0,Y 277.218,Z 244.952,A -85,B 0,C 180,E1 -17595.223,E2 -17595.223} C_VEL
LIN {X 0,Y 277.223,Z 244.951,A -85,B 0,C 180,E1 -17599.512,E2 -17599.512} C_VEL
LIN {X 0,Y 277.266,Z 244.948,A -85,B 0,C 180,E1 -17602.53,E2 -17602.53} C_VEL
LIN {X 0,Y 277.248,Z 244.945,A -85,B 0,C 180,E1 -17606.104,E2 -17606.104} C_VEL
LIN {X 0,Y 277.237,Z 244.943,A -85,B 0,C 180,E1 -17610.476,E2 -17610.476} C_VEL
LIN {X 0,Y 277.357,Z 244.936,A -85,B 0,C 180,E1 -17612.864,E2 -17612.864} C_VEL
LIN {X 0,Y 277.285,Z 244.929,A -85,B 0,C 180,E1 -17616.77,E2 -17616.77} C_VEL
LIN {X 0,Y 276.587,Z 245.014,A -85,B 0,C 180,E1 -17617.983,E2 -17617.983} C_VEL
LIN {X 0,Y 273.716,Z 245.379,A -85,B 0,C 180,E1 -17619.958,E2 -17619.958} C_VEL
LIN {X 0,Y 271.341,Z 245.68,A -85,B 0,C 180,E1 -17621.563,E2 -17621.563} C_VEL
LIN {X 0,Y 270.385,Z 245.804,A -85,B 0,C 180,E1 -17622.807,E2 -17622.807} C_VEL
LIN {X 0,Y 270.34,Z 245.805,A -85,B 0,C 180,E1 -17623.228,E2 -17623.228} C_VEL
LIN {X 0,Y 270.359,Z 245.798,A -85,B 0,C 180,E1 -17626.47,E2 -17626.47} C_VEL
LIN {X 0,Y 270.528,Z 245.777,A -85,B 0,C 180,E1 -17631.032,E2 -17631.032} C_VEL
LIN {X 0,Y 270.518,Z 245.784,A -85,B 0,C 180,E1 -17634.035,E2 -17634.035} C_VEL
LIN {X 0,Y 270.786,Z 245.75,A -85,B 0,C 180,E1 -17638.513,E2 -17638.513} C_VEL
LIN {X 0,Y 270.786,Z 245.752,A -85,B 0,C 180,E1 -17641.487,E2 -17641.487} C_VEL
LIN {X 0,Y 270.612,Z 245.774,A -85,B 0,C 180,E1 -17647.461,E2 -17647.461} C_VEL
LIN {X 0,Y 270.442,Z 245.791,A -85,B 0,C 180,E1 -17650.481,E2 -17650.481} C_VEL
LIN {X 0,Y 270.368,Z 245.805,A -85,B 0,C 180,E1 -17655.067,E2 -17655.067} C_VEL
LIN {X 0,Y 270.251,Z 245.815,A -85,B 0,C 180,E1 -17659.759,E2 -17659.759} C_VEL
LIN {X 0,Y 270.226,Z 245.82,A -85,B 0,C 180,E1 -17664.59,E2 -17664.59} C_VEL
LIN {X 0,Y 270.203,Z 245.826,A -85,B 0,C 180,E1 -17667.916,E2 -17667.916} C_VEL
LIN {X 0,Y 270.173,Z 245.828,A -85,B 0,C 180,E1 -17671.35,E2 -17671.35} C_VEL
LIN {X 0,Y 270.201,Z 245.825,A -85,B 0,C 180,E1 -17674.906,E2 -17674.906} C_VEL
LIN {X 0,Y 270.198,Z 245.827,A -85,B 0,C 180,E1 -17678.71,E2 -17678.71} C_VEL
LIN {X 0,Y 270.157,Z 245.832,A -85,B 0,C 180,E1 -17683.247,E2 -17683.247} C_VEL
LIN {X 0,Y 270.172,Z 245.826,A -85,B 0,C 180,E1 -17687.442,E2 -17687.442} C_VEL
LIN {X 0,Y 270.207,Z 245.825,A -85,B 0,C 180,E1 -17691.374,E2 -17691.374} C_VEL
LIN {X 0,Y 270.223,Z 245.826,A -85,B 0,C 180,E1 -17695.098,E2 -17695.098} C_VEL
LIN {X 0,Y 270.262,Z 246.004,A -85,B 0,C 180,E1 -17696.036,E2 -17696.036} C_VEL
LIN {X 0,Y 272.588,Z 256.546,A -85,B 0,C 180,E1 -17699.817,E2 -17699.817} C_VEL
LIN {X 0,Y 273.892,Z 263.049,A -85,B 0,C 180,E1 -17701.983,E2 -17701.983} C_VEL
LIN {X 0,Y 277.392,Z 273.126,A -85,B 0,C 180,E1 -17702.606,E2 -17702.606} C_VEL
LIN {X 0,Y 281.968,Z 305.313,A -85,B 0,C 180,E1 -17703.911,E2 -17703.911} C_VEL
LIN {X 0,Y 282.318,Z 310.601,A -85,B 0,C 180,E1 -17704.086,E2 -17704.086} C_VEL
LIN {X 0,Y 280.567,Z 371.688,A -85,B 0,C 180,E1 -17705.636,E2 -17705.636} C_VEL
LIN {X 0,Y 279.678,Z 384.837,A -85,B 0,C 180,E1 -17706.244,E2 -17706.244} C_VEL
LIN {X 0,Y 278.512,Z 396.946,A -85,B 0,C 180,E1 -17707.073,E2 -17707.073} C_VEL
LIN {X 0,Y 277.059,Z 409.165,A -85,B 0,C 180,E1 -17708.224,E2 -17708.224} C_VEL
LIN {X 0,Y 275.396,Z 420.755,A -85,B 0,C 180,E1 -17709.653,E2 -17709.653} C_VEL
LIN {X 0,Y 273.75,Z 431.192,A -85,B 0,C 180,E1 -17711.282,E2 -17711.282} C_VEL
LIN {X 0,Y 272.349,Z 441.074,A -85,B 0,C 180,E1 -17713.241,E2 -17713.241} C_VEL
LIN {X 0,Y 270.942,Z 449.642,A -85,B 0,C 180,E1 -17715.35,E2 -17715.35} C_VEL
LIN {X 0,Y 269.703,Z 456.936,A -85,B 0,C 180,E1 -17717.586,E2 -17717.586} C_VEL
LIN {X 0,Y 269.073,Z 461.867,A -85,B 0,C 180,E1 -17719.465,E2 -17719.465} C_VEL
LIN {X 0,Y 268.537,Z 466.651,A -85,B 0,C 180,E1 -17721.724,E2 -17721.724} C_VEL
LIN {X 0,Y 268.248,Z 470.305,A -85,B 0,C 180,E1 -17723.984,E2 -17723.984} C_VEL
LIN {X 0,Y 268.162,Z 472.19,A -85,B 0,C 180,E1 -17725.491,E2 -17725.491} C_VEL
LIN {X 0,Y 268.168,Z 473.608,A -85,B 0,C 180,E1 -17726.996,E2 -17726.996} C_VEL
LIN {X 0,Y 268.189,Z 474.613,A -85,B 0,C 180,E1 -17728.498,E2 -17728.498} C_VEL
LIN {X 0,Y 268.201,Z 475.225,A -85,B 0,C 180,E1 -17730,E2 -17730} C_VEL
LIN {X 0,Y 268.181,Z 475.447,A -85,B 0,C 180,E1 -17731.502,E2 -17731.502} C_VEL
LIN {X 0,Y 268.157,Z 475.238,A -85,B 0,C 180,E1 -17733.005,E2 -17733.005} C_VEL
LIN {X 0,Y 268.227,Z 473.64,A -85,B 0,C 180,E1 -17736.016,E2 -17736.016} C_VEL
LIN {X 0,Y 268.452,Z 472.258,A -85,B 0,C 180,E1 -17737.522,E2 -17737.522} C_VEL
LIN {X 0,Y 268.996,Z 469.348,A -85,B 0,C 180,E1 -17739.778,E2 -17739.778} C_VEL
LIN {X 0,Y 269.868,Z 465.422,A -85,B 0,C 180,E1 -17742.025,E2 -17742.025} C_VEL
LIN {X 0,Y 271.072,Z 460.38,A -85,B 0,C 180,E1 -17744.259,E2 -17744.259} C_VEL
LIN {X 0,Y 272.797,Z 454.061,A -85,B 0,C 180,E1 -17746.463,E2 -17746.463} C_VEL
LIN {X 0,Y 274.805,Z 446.005,A -85,B 0,C 180,E1 -17748.685,E2 -17748.685} C_VEL
LIN {X 0,Y 276.972,Z 436.361,A -85,B 0,C 180,E1 -17750.808,E2 -17750.808} C_VEL
LIN {X 0,Y 279.369,Z 426.146,A -85,B 0,C 180,E1 -17752.559,E2 -17752.559} C_VEL
LIN {X 0,Y 281.663,Z 414.627,A -85,B 0,C 180,E1 -17754.116,E2 -17754.116} C_VEL
LIN {X 0,Y 283.709,Z 403.279,A -85,B 0,C 180,E1 -17755.297,E2 -17755.297} C_VEL
LIN {X 0,Y 285.37,Z 391.629,A -85,B 0,C 180,E1 -17756.216,E2 -17756.216} C_VEL
LIN {X 0,Y 286.682,Z 379.143,A -85,B 0,C 180,E1 -17756.921,E2 -17756.921} C_VEL
LIN {X 0,Y 287.551,Z 366.513,A -85,B 0,C 180,E1 -17757.374,E2 -17757.374} C_VEL
LIN {X 0,Y 289.324,Z 311.096,A -85,B 0,C 180,E1 -17758.744,E2 -17758.744} C_VEL
LIN {X 0,Y 284.95,Z 285.907,A -85,B 0,C 180,E1 -17760.011,E2 -17760.011} C_VEL
LIN {X 0,Y 278.019,Z 270.174,A -85,B 0,C 180,E1 -17761.399,E2 -17761.399} C_VEL
LIN {X 0,Y 274.263,Z 262.231,A -85,B 0,C 180,E1 -17762.199,E2 -17762.199} C_VEL
LIN {X 0,Y 271.99,Z 252.506,A -85,B 0,C 180,E1 -17766.004,E2 -17766.004} C_VEL
LIN {X 0,Y 270.204,Z 245.828,A -85,B 0,C 180,E1 -17768.841,E2 -17768.841} C_VEL
LIN {X 0,Y 270.166,Z 245.833,A -85,B 0,C 180,E1 -17773.249,E2 -17773.249} C_VEL
LIN {X 0,Y 270.155,Z 245.834,A -85,B 0,C 180,E1 -17777.438,E2 -17777.438} C_VEL
LIN {X 0,Y 270.208,Z 245.828,A -85,B 0,C 180,E1 -17781.374,E2 -17781.374} C_VEL
LIN {X 0,Y 270.198,Z 245.828,A -85,B 0,C 180,E1 -17785.094,E2 -17785.094} C_VEL
LIN {X 0,Y 270.185,Z 245.828,A -85,B 0,C 180,E1 -17789.136,E2 -17789.136} C_VEL
LIN {X 0,Y 270.226,Z 245.824,A -85,B 0,C 180,E1 -17792.161,E2 -17792.161} C_VEL
LIN {X 0,Y 270.231,Z 245.819,A -85,B 0,C 180,E1 -17795.541,E2 -17795.541} C_VEL
LIN {X 0,Y 270.262,Z 245.819,A -85,B 0,C 180,E1 -17800.242,E2 -17800.242} C_VEL
LIN {X 0,Y 270.374,Z 245.803,A -85,B 0,C 180,E1 -17804.934,E2 -17804.934} C_VEL
LIN {X 0,Y 270.443,Z 245.793,A -85,B 0,C 180,E1 -17809.519,E2 -17809.519} C_VEL
LIN {X 0,Y 270.609,Z 245.766,A -85,B 0,C 180,E1 -17812.539,E2 -17812.539} C_VEL
LIN {X 0,Y 270.783,Z 245.743,A -85,B 0,C 180,E1 -17818.513,E2 -17818.513} C_VEL
LIN {X 0,Y 270.785,Z 245.751,A -85,B 0,C 180,E1 -17821.487,E2 -17821.487} C_VEL
LIN {X 0,Y 270.567,Z 245.772,A -85,B 0,C 180,E1 -17827.463,E2 -17827.463} C_VEL
LIN {X 0,Y 270.411,Z 245.8,A -85,B 0,C 180,E1 -17830.482,E2 -17830.482} C_VEL
LIN {X 0,Y 270.378,Z 245.802,A -85,B 0,C 180,E1 -17835.066,E2 -17835.066} C_VEL
LIN {X 0,Y 270.298,Z 245.813,A -85,B 0,C 180,E1 -17839.756,E2 -17839.756} C_VEL
LIN {X 0,Y 270.275,Z 245.816,A -85,B 0,C 180,E1 -17844.586,E2 -17844.586} C_VEL
LIN {X 0,Y 270.273,Z 245.819,A -85,B 0,C 180,E1 -17847.909,E2 -17847.909} C_VEL
LIN {X 0,Y 270.185,Z 245.828,A -85,B 0,C 180,E1 -17851.348,E2 -17851.348} C_VEL
LIN {X 0,Y 270.216,Z 245.826,A -85,B 0,C 180,E1 -17854.904,E2 -17854.904} C_VEL
LIN {X 0,Y 270.224,Z 245.822,A -85,B 0,C 180,E1 -17858.717,E2 -17858.717} C_VEL
LIN {X 0,Y 270.173,Z 245.831,A -85,B 0,C 180,E1 -17863.251,E2 -17863.251} C_VEL
LIN {X 0,Y 270.166,Z 245.826,A -85,B 0,C 180,E1 -17867.441,E2 -17867.441} C_VEL
LIN {X 0,Y 270.196,Z 246.029,A -85,B 0,C 180,E1 -17869.697,E2 -17869.697} C_VEL
LIN {X 0,Y 271.379,Z 250.168,A -85,B 0,C 180,E1 -17871.45,E2 -17871.45} C_VEL
LIN {X 0,Y 281.002,Z 268.737,A -85,B 0,C 180,E1 -17873.39,E2 -17873.39} C_VEL
LIN {X 0,Y 288.196,Z 284.874,A -85,B 0,C 180,E1 -17874.795,E2 -17874.795} C_VEL
LIN {X 0,Y 290.137,Z 289.642,A -85,B 0,C 180,E1 -17875.17,E2 -17875.17} C_VEL
LIN {X 0,Y 287.766,Z 357.048,A -85,B 0,C 180,E1 -17876.839,E2 -17876.839} C_VEL
LIN {X 0,Y 286.789,Z 370.193,A -85,B 0,C 180,E1 -17877.428,E2 -17877.428} C_VEL
LIN {X 0,Y 285.393,Z 382.479,A -85,B 0,C 180,E1 -17878.239,E2 -17878.239} C_VEL
LIN {X 0,Y 283.713,Z 394.014,A -85,B 0,C 180,E1 -17879.275,E2 -17879.275} C_VEL
LIN {X 0,Y 281.709,Z 405.625,A -85,B 0,C 180,E1 -17880.657,E2 -17880.657} C_VEL
LIN {X 0,Y 279.759,Z 415.293,A -85,B 0,C 180,E1 -17882.103,E2 -17882.103} C_VEL
LIN {X 0,Y 277.62,Z 424.076,A -85,B 0,C 180,E1 -17883.703,E2 -17883.703} C_VEL
LIN {X 0,Y 275.742,Z 432.143,A -85,B 0,C 180,E1 -17885.533,E2 -17885.533} C_VEL
LIN {X 0,Y 273.763,Z 439.886,A -85,B 0,C 180,E1 -17887.704,E2 -17887.704} C_VEL
LIN {X 0,Y 272.328,Z 445.346,A -85,B 0,C 180,E1 -17889.611,E2 -17889.611} C_VEL
LIN {X 0,Y 270.894,Z 450.516,A -85,B 0,C 180,E1 -17891.861,E2 -17891.861} C_VEL
LIN {X 0,Y 269.638,Z 455.268,A -85,B 0,C 180,E1 -17894.665,E2 -17894.665} C_VEL
LIN {X 0,Y 269.032,Z 457.447,A -85,B 0,C 180,E1 -17896.402,E2 -17896.402} C_VEL
LIN {X 0,Y 268.623,Z 458.842,A -85,B 0,C 180,E1 -17897.918,E2 -17897.918} C_VEL
LIN {X 0,Y 268.198,Z 460.425,A -85,B 0,C 180,E1 -17900.954,E2 -17900.954} C_VEL
LIN {X 0,Y 268.155,Z 460.631,A -85,B 0,C 180,E1 -17902.47,E2 -17902.47} C_VEL
LIN {X 0,Y 268.172,Z 460.142,A -85,B 0,C 180,E1 -17904.793,E2 -17904.793} C_VEL
LIN {X 0,Y 268.234,Z 458.796,A -85,B 0,C 180,E1 -17906.996,E2 -17906.996} C_VEL
LIN {X 0,Y 268.299,Z 457.405,A -85,B 0,C 180,E1 -17908.499,E2 -17908.499} C_VEL
LIN {X 0,Y 268.605,Z 454.492,A -85,B 0,C 180,E1 -17910.75,E2 -17910.75} C_VEL
LIN {X 0,Y 269.085,Z 450.556,A -85,B 0,C 180,E1 -17912.994,E2 -17912.994} C_VEL
LIN {X 0,Y 269.907,Z 445.484,A -85,B 0,C 180,E1 -17915.229,E2 -17915.229} C_VEL
LIN {X 0,Y 270.884,Z 439.109,A -85,B 0,C 180,E1 -17917.454,E2 -17917.454} C_VEL
LIN {X 0,Y 272.287,Z 431.155,A -85,B 0,C 180,E1 -17919.658,E2 -17919.658} C_VEL
LIN {X 0,Y 273.732,Z 423.045,A -85,B 0,C 180,E1 -17921.477,E2 -17921.477} C_VEL
LIN {X 0,Y 275.226,Z 413.176,A -85,B 0,C 180,E1 -17923.286,E2 -17923.286} C_VEL
LIN {X 0,Y 276.771,Z 402.38,A -85,B 0,C 180,E1 -17924.851,E2 -17924.851} C_VEL
LIN {X 0,Y 278.181,Z 391.117,A -85,B 0,C 180,E1 -17926.135,E2 -17926.135} C_VEL
LIN {X 0,Y 279.444,Z 379.048,A -85,B 0,C 180,E1 -17927.188,E2 -17927.188} C_VEL
LIN {X 0,Y 280.346,Z 366.512,A -85,B 0,C 180,E1 -17927.979,E2 -17927.979} C_VEL
LIN {X 0,Y 280.945,Z 353.394,A -85,B 0,C 180,E1 -17928.505,E2 -17928.505} C_VEL
LIN {X 0,Y 282.899,Z 283.734,A -85,B 0,C 180,E1 -17930.24,E2 -17930.24} C_VEL
LIN {X 0,Y 281.503,Z 276.297,A -85,B 0,C 180,E1 -17930.57,E2 -17930.57} C_VEL
LIN {X 0,Y 274.891,Z 258.611,A -85,B 0,C 180,E1 -17931.691,E2 -17931.691} C_VEL
LIN {X 0,Y 271.092,Z 249.525,A -85,B 0,C 180,E1 -17932.344,E2 -17932.344} C_VEL
LIN {X 0,Y 270.276,Z 245.819,A -85,B 0,C 180,E1 -17933.769,E2 -17933.769} C_VEL
LIN {X 0,Y 270.211,Z 245.826,A -85,B 0,C 180,E1 -17937.915,E2 -17937.915} C_VEL
LIN {X 0,Y 270.175,Z 245.83,A -85,B 0,C 180,E1 -17941.349,E2 -17941.349} C_VEL
LIN {X 0,Y 270.204,Z 245.828,A -85,B 0,C 180,E1 -17944.905,E2 -17944.905} C_VEL
LIN {X 0,Y 270.199,Z 245.829,A -85,B 0,C 180,E1 -17948.71,E2 -17948.71} C_VEL
LIN {X 0,Y 270.173,Z 245.829,A -85,B 0,C 180,E1 -17953.25,E2 -17953.25} C_VEL
LIN {X 0,Y 270.176,Z 245.829,A -85,B 0,C 180,E1 -17957.442,E2 -17957.442} C_VEL
LIN {X 0,Y 270.208,Z 245.823,A -85,B 0,C 180,E1 -17961.374,E2 -17961.374} C_VEL
LIN {X 0,Y 270.202,Z 245.823,A -85,B 0,C 180,E1 -17965.094,E2 -17965.094} C_VEL
LIN {X 0,Y 270.201,Z 245.821,A -85,B 0,C 180,E1 -17969.13,E2 -17969.13} C_VEL
LIN {X 0,Y 270.264,Z 245.818,A -85,B 0,C 180,E1 -17972.146,E2 -17972.146} C_VEL
LIN {X 0,Y 270.278,Z 245.809,A -85,B 0,C 180,E1 -17975.519,E2 -17975.519} C_VEL
LIN {X 0,Y 270.303,Z 245.806,A -85,B 0,C 180,E1 -17980.244,E2 -17980.244} C_VEL
LIN {X 0,Y 270.34,Z 245.805,A -85,B 0,C 180,E1 -17983.228,E2 -17983.228} C_VEL
LIN {X 0,Y 270.084,Z 245.841,A -85,B 0,C 180,E1 -17984.06,E2 -17984.06} C_VEL
LIN {X 0,Y 268.769,Z 246.003,A -85,B 0,C 180,E1 -17985.288,E2 -17985.288} C_VEL
LIN {X 0,Y 264.439,Z 246.526,A -85,B 0,C 180,E1 -17988.146,E2 -17988.146} C_VEL
LIN {X 0,Y 263.441,Z 246.649,A -85,B 0,C 180,E1 -17989.425,E2 -17989.425} C_VEL
LIN {X 0,Y 263.39,Z 246.655,A -85,B 0,C 180,E1 -17989.858,E2 -17989.858} C_VEL
LIN {X 0,Y 263.529,Z 246.651,A -85,B 0,C 180,E1 -17992.337,E2 -17992.337} C_VEL
LIN {X 0,Y 263.75,Z 246.626,A -85,B 0,C 180,E1 -17998.473,E2 -17998.473} C_VEL
LIN {X 0,Y 263.75,Z 246.628,A -85,B 0,C 180,E1 -18001.527,E2 -18001.527} C_VEL
LIN {X 0,Y 263.574,Z 246.651,A -85,B 0,C 180,E1 -18007.661,E2 -18007.661} C_VEL
LIN {X 0,Y 263.374,Z 246.669,A -85,B 0,C 180,E1 -18010.765,E2 -18010.765} C_VEL
LIN {X 0,Y 263.31,Z 246.683,A -85,B 0,C 180,E1 -18015.48,E2 -18015.48} C_VEL
LIN {X 0,Y 263.235,Z 246.691,A -85,B 0,C 180,E1 -18020.309,E2 -18020.309} C_VEL
LIN {X 0,Y 263.17,Z 246.698,A -85,B 0,C 180,E1 -18025.295,E2 -18025.295} C_VEL
LIN {X 0,Y 263.136,Z 246.707,A -85,B 0,C 180,E1 -18028.735,E2 -18028.735} C_VEL
LIN {X 0,Y 263.128,Z 246.708,A -85,B 0,C 180,E1 -18032.289,E2 -18032.289} C_VEL
LIN {X 0,Y 263.18,Z 246.703,A -85,B 0,C 180,E1 -18036.762,E2 -18036.762} C_VEL
LIN {X 0,Y 263.091,Z 246.711,A -85,B 0,C 180,E1 -18039.875,E2 -18039.875} C_VEL
LIN {X 0,Y 263.102,Z 246.711,A -85,B 0,C 180,E1 -18043.989,E2 -18043.989} C_VEL
LIN {X 0,Y 263.124,Z 246.703,A -85,B 0,C 180,E1 -18048.107,E2 -18048.107} C_VEL
LIN {X 0,Y 263.166,Z 246.704,A -85,B 0,C 180,E1 -18052.104,E2 -18052.104} C_VEL
LIN {X 0,Y 263.207,Z 246.735,A -85,B 0,C 180,E1 -18055.432,E2 -18055.432} C_VEL
LIN {X 0,Y 265.51,Z 257.371,A -85,B 0,C 180,E1 -18059.367,E2 -18059.367} C_VEL
LIN {X 0,Y 266.606,Z 262.662,A -85,B 0,C 180,E1 -18061.23,E2 -18061.23} C_VEL
LIN {X 0,Y 271.016,Z 274.734,A -85,B 0,C 180,E1 -18062.032,E2 -18062.032} C_VEL
LIN {X 0,Y 275.12,Z 303.329,A -85,B 0,C 180,E1 -18063.238,E2 -18063.238} C_VEL
LIN {X 0,Y 275.83,Z 309.205,A -85,B 0,C 180,E1 -18063.468,E2 -18063.468} C_VEL
LIN {X 0,Y 274.022,Z 371.021,A -85,B 0,C 180,E1 -18065.066,E2 -18065.066} C_VEL
LIN {X 0,Y 273.1,Z 384.327,A -85,B 0,C 180,E1 -18065.685,E2 -18065.685} C_VEL
LIN {X 0,Y 271.844,Z 397.088,A -85,B 0,C 180,E1 -18066.579,E2 -18066.579} C_VEL
LIN {X 0,Y 270.441,Z 408.408,A -85,B 0,C 180,E1 -18067.663,E2 -18067.663} C_VEL
LIN {X 0,Y 268.697,Z 420.1,A -85,B 0,C 180,E1 -18069.122,E2 -18069.122} C_VEL
LIN {X 0,Y 266.958,Z 430.613,A -85,B 0,C 180,E1 -18070.787,E2 -18070.787} C_VEL
LIN {X 0,Y 265.578,Z 440.247,A -85,B 0,C 180,E1 -18072.718,E2 -18072.718} C_VEL
LIN {X 0,Y 264.039,Z 449.206,A -85,B 0,C 180,E1 -18074.959,E2 -18074.959} C_VEL
LIN {X 0,Y 262.745,Z 456.542,A -85,B 0,C 180,E1 -18077.251,E2 -18077.251} C_VEL
LIN {X 0,Y 262.051,Z 461.509,A -85,B 0,C 180,E1 -18079.179,E2 -18079.179} C_VEL
LIN {X 0,Y 261.499,Z 466.328,A -85,B 0,C 180,E1 -18081.5,E2 -18081.5} C_VEL
LIN {X 0,Y 261.166,Z 470.014,A -85,B 0,C 180,E1 -18083.821,E2 -18083.821} C_VEL
LIN {X 0,Y 261.067,Z 471.916,A -85,B 0,C 180,E1 -18085.368,E2 -18085.368} C_VEL
LIN {X 0,Y 261.083,Z 473.362,A -85,B 0,C 180,E1 -18086.914,E2 -18086.914} C_VEL
LIN {X 0,Y 261.116,Z 474.382,A -85,B 0,C 180,E1 -18088.458,E2 -18088.458} C_VEL
LIN {X 0,Y 261.127,Z 475.008,A -85,B 0,C 180,E1 -18090,E2 -18090} C_VEL
LIN {X 0,Y 261.108,Z 475.246,A -85,B 0,C 180,E1 -18091.542,E2 -18091.542} C_VEL
LIN {X 0,Y 261.053,Z 475.063,A -85,B 0,C 180,E1 -18093.087,E2 -18093.087} C_VEL
LIN {X 0,Y 261.154,Z 473.492,A -85,B 0,C 180,E1 -18096.18,E2 -18096.18} C_VEL
LIN {X 0,Y 261.382,Z 472.124,A -85,B 0,C 180,E1 -18097.726,E2 -18097.726} C_VEL
LIN {X 0,Y 261.992,Z 469.245,A -85,B 0,C 180,E1 -18100.042,E2 -18100.042} C_VEL
LIN {X 0,Y 262.879,Z 465.35,A -85,B 0,C 180,E1 -18102.35,E2 -18102.35} C_VEL
LIN {X 0,Y 264.188,Z 460.342,A -85,B 0,C 180,E1 -18104.639,E2 -18104.639} C_VEL
LIN {X 0,Y 265.976,Z 454.068,A -85,B 0,C 180,E1 -18106.897,E2 -18106.897} C_VEL
LIN {X 0,Y 267.946,Z 446.615,A -85,B 0,C 180,E1 -18109.036,E2 -18109.036} C_VEL
LIN {X 0,Y 269.911,Z 438.26,A -85,B 0,C 180,E1 -18110.979,E2 -18110.979} C_VEL
LIN {X 0,Y 272.323,Z 428.546,A -85,B 0,C 180,E1 -18112.775,E2 -18112.775} C_VEL
LIN {X 0,Y 274.703,Z 417.758,A -85,B 0,C 180,E1 -18114.365,E2 -18114.365} C_VEL
LIN {X 0,Y 276.729,Z 407.238,A -85,B 0,C 180,E1 -18115.578,E2 -18115.578} C_VEL
LIN {X 0,Y 278.726,Z 394.588,A -85,B 0,C 180,E1 -18116.688,E2 -18116.688} C_VEL
LIN {X 0,Y 280.214,Z 381.953,A -85,B 0,C 180,E1 -18117.493,E2 -18117.493} C_VEL
LIN {X 0,Y 281.214,Z 369.95,A -85,B 0,C 180,E1 -18117.994,E2 -18117.994} C_VEL
LIN {X 0,Y 283.199,Z 311.88,A -85,B 0,C 180,E1 -18119.472,E2 -18119.472} C_VEL
LIN {X 0,Y 279.155,Z 288.428,A -85,B 0,C 180,E1 -18120.692,E2 -18120.692} C_VEL
LIN {X 0,Y 272.381,Z 273.177,A -85,B 0,C 180,E1 -18122.102,E2 -18122.102} C_VEL
LIN {X 0,Y 268.151,Z 264.721,A -85,B 0,C 180,E1 -18122.998,E2 -18122.998} C_VEL
LIN {X 0,Y 266.988,Z 261.881,A -85,B 0,C 180,E1 -18123.327,E2 -18123.327} C_VEL
LIN {X 0,Y 264.726,Z 252.413,A -85,B 0,C 180,E1 -18127.208,E2 -18127.208} C_VEL
LIN {X 0,Y 263.149,Z 246.707,A -85,B 0,C 180,E1 -18129.771,E2 -18129.771} C_VEL
LIN {X 0,Y 263.123,Z 246.711,A -85,B 0,C 180,E1 -18133.984,E2 -18133.984} C_VEL
LIN {X 0,Y 263.11,Z 246.711,A -85,B 0,C 180,E1 -18138.41,E2 -18138.41} C_VEL
LIN {X 0,Y 263.157,Z 246.702,A -85,B 0,C 180,E1 -18142.103,E2 -18142.103} C_VEL
LIN {X 0,Y 263.152,Z 246.699,A -85,B 0,C 180,E1 -18145.886,E2 -18145.886} C_VEL
LIN {X 0,Y 263.127,Z 246.703,A -85,B 0,C 180,E1 -18149.504,E2 -18149.504} C_VEL
LIN {X 0,Y 263.151,Z 246.706,A -85,B 0,C 180,E1 -18152.998,E2 -18152.998} C_VEL
LIN {X 0,Y 263.149,Z 246.705,A -85,B 0,C 180,E1 -18156.384,E2 -18156.384} C_VEL
LIN {X 0,Y 263.239,Z 246.689,A -85,B 0,C 180,E1 -18159.691,E2 -18159.691} C_VEL
LIN {X 0,Y 263.315,Z 246.681,A -85,B 0,C 180,E1 -18164.52,E2 -18164.52} C_VEL
LIN {X 0,Y 263.375,Z 246.67,A -85,B 0,C 180,E1 -18169.235,E2 -18169.235} C_VEL
LIN {X 0,Y 263.571,Z 246.643,A -85,B 0,C 180,E1 -18172.338,E2 -18172.338} C_VEL
LIN {X 0,Y 263.748,Z 246.619,A -85,B 0,C 180,E1 -18178.473,E2 -18178.473} C_VEL
LIN {X 0,Y 263.75,Z 246.627,A -85,B 0,C 180,E1 -18181.527,E2 -18181.527} C_VEL
LIN {X 0,Y 263.53,Z 246.647,A -85,B 0,C 180,E1 -18187.663,E2 -18187.663} C_VEL
LIN {X 0,Y 263.351,Z 246.68,A -85,B 0,C 180,E1 -18190.767,E2 -18190.767} C_VEL
LIN {X 0,Y 263.325,Z 246.684,A -85,B 0,C 180,E1 -18195.48,E2 -18195.48} C_VEL
LIN {X 0,Y 263.263,Z 246.689,A -85,B 0,C 180,E1 -18200.307,E2 -18200.307} C_VEL
LIN {X 0,Y 263.209,Z 246.694,A -85,B 0,C 180,E1 -18205.292,E2 -18205.292} C_VEL
LIN {X 0,Y 263.18,Z 246.701,A -85,B 0,C 180,E1 -18208.73,E2 -18208.73} C_VEL
LIN {X 0,Y 263.135,Z 246.707,A -85,B 0,C 180,E1 -18212.288,E2 -18212.288} C_VEL
LIN {X 0,Y 263.189,Z 246.696,A -85,B 0,C 180,E1 -18215.978,E2 -18215.978} C_VEL
LIN {X 0,Y 263.117,Z 246.71,A -85,B 0,C 180,E1 -18219.871,E2 -18219.871} C_VEL
LIN {X 0,Y 263.13,Z 246.708,A -85,B 0,C 180,E1 -18223.983,E2 -18223.983} C_VEL
LIN {X 0,Y 263.117,Z 246.711,A -85,B 0,C 180,E1 -18228.105,E2 -18228.105} C_VEL
LIN {X 0,Y 263.138,Z 246.903,A -85,B 0,C 180,E1 -18228.793,E2 -18228.793} C_VEL
LIN {X 0,Y 264.168,Z 250.53,A -85,B 0,C 180,E1 -18230.343,E2 -18230.343} C_VEL
LIN {X 0,Y 272.998,Z 266.946,A -85,B 0,C 180,E1 -18232.219,E2 -18232.219} C_VEL
LIN {X 0,Y 280.521,Z 282.96,A -85,B 0,C 180,E1 -18233.753,E2 -18233.753} C_VEL
LIN {X 0,Y 284.033,Z 291.451,A -85,B 0,C 180,E1 -18234.462,E2 -18234.462} C_VEL
LIN {X 0,Y 281.598,Z 357.446,A -85,B 0,C 180,E1 -18236.129,E2 -18236.129} C_VEL
LIN {X 0,Y 280.614,Z 370.451,A -85,B 0,C 180,E1 -18236.726,E2 -18236.726} C_VEL
LIN {X 0,Y 279.168,Z 382.721,A -85,B 0,C 180,E1 -18237.552,E2 -18237.552} C_VEL
LIN {X 0,Y 277.27,Z 395.05,A -85,B 0,C 180,E1 -18238.693,E2 -18238.693} C_VEL
LIN {X 0,Y 275.126,Z 406.973,A -85,B 0,C 180,E1 -18240.171,E2 -18240.171} C_VEL
LIN {X 0,Y 272.938,Z 417.129,A -85,B 0,C 180,E1 -18241.761,E2 -18241.761} C_VEL
LIN {X 0,Y 270.757,Z 425.632,A -85,B 0,C 180,E1 -18243.4,E2 -18243.4} C_VEL
LIN {X 0,Y 268.442,Z 434.816,A -85,B 0,C 180,E1 -18245.648,E2 -18245.648} C_VEL
LIN {X 0,Y 266.622,Z 441.402,A -85,B 0,C 180,E1 -18247.652,E2 -18247.652} C_VEL
LIN {X 0,Y 265.006,Z 447.161,A -85,B 0,C 180,E1 -18249.833,E2 -18249.833} C_VEL
LIN {X 0,Y 263.628,Z 451.972,A -85,B 0,C 180,E1 -18252.147,E2 -18252.147} C_VEL
LIN {X 0,Y 262.628,Z 455.647,A -85,B 0,C 180,E1 -18254.478,E2 -18254.478} C_VEL
LIN {X 0,Y 262.041,Z 457.538,A -85,B 0,C 180,E1 -18256.032,E2 -18256.032} C_VEL
LIN {X 0,Y 261.597,Z 458.972,A -85,B 0,C 180,E1 -18257.589,E2 -18257.589} C_VEL
LIN {X 0,Y 261.129,Z 460.594,A -85,B 0,C 180,E1 -18260.707,E2 -18260.707} C_VEL
LIN {X 0,Y 261.065,Z 460.825,A -85,B 0,C 180,E1 -18262.264,E2 -18262.264} C_VEL
LIN {X 0,Y 261.087,Z 460.295,A -85,B 0,C 180,E1 -18264.863,E2 -18264.863} C_VEL
LIN {X 0,Y 261.142,Z 459.06,A -85,B 0,C 180,E1 -18266.914,E2 -18266.914} C_VEL
LIN {X 0,Y 261.22,Z 457.696,A -85,B 0,C 180,E1 -18268.458,E2 -18268.458} C_VEL
LIN {X 0,Y 261.511,Z 454.819,A -85,B 0,C 180,E1 -18270.77,E2 -18270.77} C_VEL
LIN {X 0,Y 262.005,Z 450.926,A -85,B 0,C 180,E1 -18273.075,E2 -18273.075} C_VEL
LIN {X 0,Y 262.846,Z 445.905,A -85,B 0,C 180,E1 -18275.37,E2 -18275.37} C_VEL
LIN {X 0,Y 263.863,Z 439.602,A -85,B 0,C 180,E1 -18277.653,E2 -18277.653} C_VEL
LIN {X 0,Y 265.309,Z 431.712,A -85,B 0,C 180,E1 -18279.915,E2 -18279.915} C_VEL
LIN {X 0,Y 266.815,Z 423.673,A -85,B 0,C 180,E1 -18281.779,E2 -18281.779} C_VEL
LIN {X 0,Y 268.356,Z 413.89,A -85,B 0,C 180,E1 -18283.633,E2 -18283.633} C_VEL
LIN {X 0,Y 269.824,Z 404.272,A -85,B 0,C 180,E1 -18285.098,E2 -18285.098} C_VEL
LIN {X 0,Y 271.268,Z 393.471,A -85,B 0,C 180,E1 -18286.414,E2 -18286.414} C_VEL
LIN {X 0,Y 272.61,Z 381.456,A -85,B 0,C 180,E1 -18287.536,E2 -18287.536} C_VEL
LIN {X 0,Y 273.655,Z 368.318,A -85,B 0,C 180,E1 -18288.434,E2 -18288.434} C_VEL
LIN {X 0,Y 274.272,Z 356.445,A -85,B 0,C 180,E1 -18288.972,E2 -18288.972} C_VEL
LIN {X 0,Y 276.369,Z 284.522,A -85,B 0,C 180,E1 -18290.819,E2 -18290.819} C_VEL
LIN {X 0,Y 275.024,Z 277.878,A -85,B 0,C 180,E1 -18291.133,E2 -18291.133} C_VEL
LIN {X 0,Y 269.055,Z 261.97,A -85,B 0,C 180,E1 -18292.182,E2 -18292.182} C_VEL
LIN {X 0,Y 263.867,Z 249.691,A -85,B 0,C 180,E1 -18293.119,E2 -18293.119} C_VEL
LIN {X 0,Y 263.203,Z 246.7,A -85,B 0,C 180,E1 -18294.299,E2 -18294.299} C_VEL
LIN {X 0,Y 263.14,Z 246.709,A -85,B 0,C 180,E1 -18298.734,E2 -18298.734} C_VEL
LIN {X 0,Y 263.13,Z 246.709,A -85,B 0,C 180,E1 -18302.289,E2 -18302.289} C_VEL
LIN {X 0,Y 263.185,Z 246.702,A -85,B 0,C 180,E1 -18306.763,E2 -18306.763} C_VEL
LIN {X 0,Y 263.127,Z 246.706,A -85,B 0,C 180,E1 -18311.593,E2 -18311.593} C_VEL
LIN {X 0,Y 263.129,Z 246.707,A -85,B 0,C 180,E1 -18316.017,E2 -18316.017} C_VEL
LIN {X 0,Y 263.107,Z 246.71,A -85,B 0,C 180,E1 -18320.127,E2 -18320.127} C_VEL
LIN {X 0,Y 263.164,Z 246.703,A -85,B 0,C 180,E1 -18324.018,E2 -18324.018} C_VEL
LIN {X 0,Y 263.134,Z 246.691,A -85,B 0,C 180,E1 -18327.712,E2 -18327.712} C_VEL
LIN {X 0,Y 263.197,Z 246.697,A -85,B 0,C 180,E1 -18331.785,E2 -18331.785} C_VEL
LIN {X 0,Y 263.227,Z 246.687,A -85,B 0,C 180,E1 -18335.2,E2 -18335.2} C_VEL
LIN {X 0,Y 263.265,Z 246.68,A -85,B 0,C 180,E1 -18339.693,E2 -18339.693} C_VEL
LIN {X 0,Y 263.352,Z 246.678,A -85,B 0,C 180,E1 -18344.522,E2 -18344.522} C_VEL
LIN {X 0,Y 263.353,Z 246.659,A -85,B 0,C 180,E1 -18349.233,E2 -18349.233} C_VEL
LIN {X 0,Y 263.39,Z 246.655,A -85,B 0,C 180,E1 -18349.858,E2 -18349.858} C_VEL
LIN {X 0,Y 263.122,Z 246.694,A -85,B 0,C 180,E1 -18350.712,E2 -18350.712} C_VEL
LIN {X 0,Y 261.781,Z 246.868,A -85,B 0,C 180,E1 -18351.972,E2 -18351.972} C_VEL
LIN {X 0,Y 257.436,Z 247.416,A -85,B 0,C 180,E1 -18354.907,E2 -18354.907} C_VEL
LIN {X 0,Y 256.486,Z 247.533,A -85,B 0,C 180,E1 -18356.221,E2 -18356.221} C_VEL
LIN {X 0,Y 256.464,Z 247.531,A -85,B 0,C 180,E1 -18356.666,E2 -18356.666} C_VEL
LIN {X 0,Y 256.713,Z 247.501,A -85,B 0,C 180,E1 -18358.431,E2 -18358.431} C_VEL
LIN {X 0,Y 256.713,Z 247.505,A -85,B 0,C 180,E1 -18361.569,E2 -18361.569} C_VEL
LIN {X 0,Y 256.541,Z 247.527,A -85,B 0,C 180,E1 -18367.873,E2 -18367.873} C_VEL
LIN {X 0,Y 256.31,Z 247.548,A -85,B 0,C 180,E1 -18371.066,E2 -18371.066} C_VEL
LIN {X 0,Y 256.233,Z 247.566,A -85,B 0,C 180,E1 -18374.291,E2 -18374.291} C_VEL
LIN {X 0,Y 256.168,Z 247.568,A -85,B 0,C 180,E1 -18377.565,E2 -18377.565} C_VEL
LIN {X 0,Y 256.141,Z 247.578,A -85,B 0,C 180,E1 -18381.11,E2 -18381.11} C_VEL
LIN {X 0,Y 256.135,Z 247.574,A -85,B 0,C 180,E1 -18385.113,E2 -18385.113} C_VEL
LIN {X 0,Y 256.056,Z 247.585,A -85,B 0,C 180,E1 -18389.607,E2 -18389.607} C_VEL
LIN {X 0,Y 256.066,Z 247.586,A -85,B 0,C 180,E1 -18393.293,E2 -18393.293} C_VEL
LIN {X 0,Y 256.112,Z 247.581,A -85,B 0,C 180,E1 -18397.27,E2 -18397.27} C_VEL
LIN {X 0,Y 256.059,Z 247.588,A -85,B 0,C 180,E1 -18402.178,E2 -18402.178} C_VEL
LIN {X 0,Y 256.062,Z 247.587,A -85,B 0,C 180,E1 -18406.673,E2 -18406.673} C_VEL
LIN {X 0,Y 256.072,Z 247.587,A -85,B 0,C 180,E1 -18410.858,E2 -18410.858} C_VEL
LIN {X 0,Y 256.156,Z 247.694,A -85,B 0,C 180,E1 -18414.875,E2 -18414.875} C_VEL
LIN {X 0,Y 258.49,Z 258.193,A -85,B 0,C 180,E1 -18418.897,E2 -18418.897} C_VEL
LIN {X 0,Y 259.428,Z 262.621,A -85,B 0,C 180,E1 -18420.453,E2 -18420.453} C_VEL
LIN {X 0,Y 264.789,Z 276.961,A -85,B 0,C 180,E1 -18421.461,E2 -18421.461} C_VEL
LIN {X 0,Y 268.761,Z 305.232,A -85,B 0,C 180,E1 -18422.687,E2 -18422.687} C_VEL
LIN {X 0,Y 269.302,Z 311.42,A -85,B 0,C 180,E1 -18422.917,E2 -18422.917} C_VEL
LIN {X 0,Y 267.442,Z 371.468,A -85,B 0,C 180,E1 -18424.513,E2 -18424.513} C_VEL
LIN {X 0,Y 266.434,Z 385.329,A -85,B 0,C 180,E1 -18425.192,E2 -18425.192} C_VEL
LIN {X 0,Y 265.095,Z 398.247,A -85,B 0,C 180,E1 -18426.153,E2 -18426.153} C_VEL
LIN {X 0,Y 263.394,Z 410.825,A -85,B 0,C 180,E1 -18427.446,E2 -18427.446} C_VEL
LIN {X 0,Y 261.642,Z 422.039,A -85,B 0,C 180,E1 -18428.945,E2 -18428.945} C_VEL
LIN {X 0,Y 259.889,Z 432.108,A -85,B 0,C 180,E1 -18430.654,E2 -18430.654} C_VEL
LIN {X 0,Y 258.494,Z 441.243,A -85,B 0,C 180,E1 -18432.598,E2 -18432.598} C_VEL
LIN {X 0,Y 256.904,Z 450.133,A -85,B 0,C 180,E1 -18434.937,E2 -18434.937} C_VEL
LIN {X 0,Y 255.579,Z 457.237,A -85,B 0,C 180,E1 -18437.292,E2 -18437.292} C_VEL
LIN {X 0,Y 254.798,Z 462.913,A -85,B 0,C 180,E1 -18439.672,E2 -18439.672} C_VEL
LIN {X 0,Y 254.305,Z 467.373,A -85,B 0,C 180,E1 -18442.057,E2 -18442.057} C_VEL
LIN {X 0,Y 253.983,Z 471.347,A -85,B 0,C 180,E1 -18444.979,E2 -18444.979} C_VEL
LIN {X 0,Y 253.98,Z 473.115,A -85,B 0,C 180,E1 -18446.828,E2 -18446.828} C_VEL
LIN {X 0,Y 254.022,Z 474.15,A -85,B 0,C 180,E1 -18448.415,E2 -18448.415} C_VEL
LIN {X 0,Y 254.054,Z 474.791,A -85,B 0,C 180,E1 -18450,E2 -18450} C_VEL
LIN {X 0,Y 254.014,Z 475.043,A -85,B 0,C 180,E1 -18451.586,E2 -18451.586} C_VEL
LIN {X 0,Y 253.953,Z 474.886,A -85,B 0,C 180,E1 -18453.173,E2 -18453.173} C_VEL
LIN {X 0,Y 253.99,Z 474.166,A -85,B 0,C 180,E1 -18455.039,E2 -18455.039} C_VEL
LIN {X 0,Y 254.335,Z 471.991,A -85,B 0,C 180,E1 -18457.942,E2 -18457.942} C_VEL
LIN {X 0,Y 254.964,Z 469.142,A -85,B 0,C 180,E1 -18460.321,E2 -18460.321} C_VEL
LIN {X 0,Y 255.903,Z 465.28,A -85,B 0,C 180,E1 -18462.692,E2 -18462.692} C_VEL
LIN {X 0,Y 257.32,Z 460.307,A -85,B 0,C 180,E1 -18465.038,E2 -18465.038} C_VEL
LIN {X 0,Y 259.168,Z 454.073,A -85,B 0,C 180,E1 -18467.355,E2 -18467.355} C_VEL
LIN {X 0,Y 261.089,Z 447.223,A -85,B 0,C 180,E1 -18469.4,E2 -18469.4} C_VEL
LIN {X 0,Y 263.305,Z 438.382,A -85,B 0,C 180,E1 -18471.531,E2 -18471.531} C_VEL
LIN {X 0,Y 265.81,Z 428.733,A -85,B 0,C 180,E1 -18473.366,E2 -18473.366} C_VEL
LIN {X 0,Y 268.26,Z 418.03,A -85,B 0,C 180,E1 -18474.989,E2 -18474.989} C_VEL
LIN {X 0,Y 270.375,Z 407.654,A -85,B 0,C 180,E1 -18476.225,E2 -18476.225} C_VEL
LIN {X 0,Y 272.436,Z 395.2,A -85,B 0,C 180,E1 -18477.355,E2 -18477.355} C_VEL
LIN {X 0,Y 274.06,Z 382.087,A -85,B 0,C 180,E1 -18478.217,E2 -18478.217} C_VEL
LIN {X 0,Y 275.2,Z 368.92,A -85,B 0,C 180,E1 -18478.766,E2 -18478.766} C_VEL
LIN {X 0,Y 277.17,Z 312.938,A -85,B 0,C 180,E1 -18480.217,E2 -18480.217} C_VEL
LIN {X 0,Y 273.497,Z 291.256,A -85,B 0,C 180,E1 -18481.379,E2 -18481.379} C_VEL
LIN {X 0,Y 266.92,Z 276.356,A -85,B 0,C 180,E1 -18482.809,E2 -18482.809} C_VEL
LIN {X 0,Y 260.994,Z 264.561,A -85,B 0,C 180,E1 -18484.128,E2 -18484.128} C_VEL
LIN {X 0,Y 259.759,Z 261.736,A -85,B 0,C 180,E1 -18484.453,E2 -18484.453} C_VEL
LIN {X 0,Y 257.839,Z 253.981,A -85,B 0,C 180,E1 -18487.771,E2 -18487.771} C_VEL
LIN {X 0,Y 256.068,Z 247.589,A -85,B 0,C 180,E1 -18490.718,E2 -18490.718} C_VEL
LIN {X 0,Y 256.054,Z 247.59,A -85,B 0,C 180,E1 -18494.469,E2 -18494.469} C_VEL
LIN {X 0,Y 256.04,Z 247.591,A -85,B 0,C 180,E1 -18498.794,E2 -18498.794} C_VEL
LIN {X 0,Y 256.126,Z 247.573,A -85,B 0,C 180,E1 -18502.867,E2 -18502.867} C_VEL
LIN {X 0,Y 256.066,Z 247.578,A -85,B 0,C 180,E1 -18506.707,E2 -18506.707} C_VEL
LIN {X 0,Y 256.058,Z 247.578,A -85,B 0,C 180,E1 -18510.393,E2 -18510.393} C_VEL
LIN {X 0,Y 256.16,Z 247.567,A -85,B 0,C 180,E1 -18514.876,E2 -18514.876} C_VEL
LIN {X 0,Y 256.149,Z 247.569,A -85,B 0,C 180,E1 -18519.103,E2 -18519.103} C_VEL
LIN {X 0,Y 256.249,Z 247.558,A -85,B 0,C 180,E1 -18524.082,E2 -18524.082} C_VEL
LIN {X 0,Y 256.291,Z 247.551,A -85,B 0,C 180,E1 -18527.328,E2 -18527.328} C_VEL
LIN {X 0,Y 256.481,Z 247.535,A -85,B 0,C 180,E1 -18530.561,E2 -18530.561} C_VEL
LIN {X 0,Y 256.485,Z 247.526,A -85,B 0,C 180,E1 -18533.708,E2 -18533.708} C_VEL
LIN {X 0,Y 256.711,Z 247.495,A -85,B 0,C 180,E1 -18538.431,E2 -18538.431} C_VEL
LIN {X 0,Y 256.713,Z 247.503,A -85,B 0,C 180,E1 -18541.569,E2 -18541.569} C_VEL
LIN {X 0,Y 256.45,Z 247.535,A -85,B 0,C 180,E1 -18546.562,E2 -18546.562} C_VEL
LIN {X 0,Y 256.428,Z 247.535,A -85,B 0,C 180,E1 -18549.465,E2 -18549.465} C_VEL
LIN {X 0,Y 256.238,Z 247.559,A -85,B 0,C 180,E1 -18554.291,E2 -18554.291} C_VEL
LIN {X 0,Y 256.185,Z 247.562,A -85,B 0,C 180,E1 -18557.564,E2 -18557.564} C_VEL
LIN {X 0,Y 256.159,Z 247.572,A -85,B 0,C 180,E1 -18561.12,E2 -18561.12} C_VEL
LIN {X 0,Y 256.19,Z 247.57,A -85,B 0,C 180,E1 -18565.139,E2 -18565.139} C_VEL
LIN {X 0,Y 256.115,Z 247.576,A -85,B 0,C 180,E1 -18569.6,E2 -18569.6} C_VEL
LIN {X 0,Y 256.087,Z 247.581,A -85,B 0,C 180,E1 -18573.29,E2 -18573.29} C_VEL
LIN {X 0,Y 256.13,Z 247.579,A -85,B 0,C 180,E1 -18577.275,E2 -18577.275} C_VEL
LIN {X 0,Y 256.059,Z 247.587,A -85,B 0,C 180,E1 -18581.203,E2 -18581.203} C_VEL
LIN {X 0,Y 256.063,Z 247.586,A -85,B 0,C 180,E1 -18585.529,E2 -18585.529} C_VEL
LIN {X 0,Y 256.085,Z 247.758,A -85,B 0,C 180,E1 -18587.816,E2 -18587.816} C_VEL
LIN {X 0,Y 256.866,Z 250.668,A -85,B 0,C 180,E1 -18589.132,E2 -18589.132} C_VEL
LIN {X 0,Y 259.198,Z 254.659,A -85,B 0,C 180,E1 -18589.667,E2 -18589.667} C_VEL
LIN {X 0,Y 267.928,Z 270.967,A -85,B 0,C 180,E1 -18591.596,E2 -18591.596} C_VEL
LIN {X 0,Y 275.113,Z 286.356,A -85,B 0,C 180,E1 -18593.122,E2 -18593.122} C_VEL
LIN {X 0,Y 277.955,Z 293.327,A -85,B 0,C 180,E1 -18593.722,E2 -18593.722} C_VEL
LIN {X 0,Y 275.505,Z 357.678,A -85,B 0,C 180,E1 -18595.382,E2 -18595.382} C_VEL
LIN {X 0,Y 274.482,Z 370.709,A -85,B 0,C 180,E1 -18595.993,E2 -18595.993} C_VEL
LIN {X 0,Y 272.995,Z 382.965,A -85,B 0,C 180,E1 -18596.834,E2 -18596.834} C_VEL
LIN {X 0,Y 271.204,Z 394.476,A -85,B 0,C 180,E1 -18597.911,E2 -18597.911} C_VEL
LIN {X 0,Y 269.219,Z 404.955,A -85,B 0,C 180,E1 -18599.183,E2 -18599.183} C_VEL
LIN {X 0,Y 267.107,Z 414.649,A -85,B 0,C 180,E1 -18600.656,E2 -18600.656} C_VEL
LIN {X 0,Y 264.805,Z 423.606,A -85,B 0,C 180,E1 -18602.325,E2 -18602.325} C_VEL
LIN {X 0,Y 262.683,Z 431.815,A -85,B 0,C 180,E1 -18604.23,E2 -18604.23} C_VEL
LIN {X 0,Y 260.443,Z 439.89,A -85,B 0,C 180,E1 -18606.562,E2 -18606.562} C_VEL
LIN {X 0,Y 258.855,Z 445.251,A -85,B 0,C 180,E1 -18608.498,E2 -18608.498} C_VEL
LIN {X 0,Y 257.211,Z 450.528,A -85,B 0,C 180,E1 -18610.859,E2 -18610.859} C_VEL
LIN {X 0,Y 256.024,Z 454.613,A -85,B 0,C 180,E1 -18613.248,E2 -18613.248} C_VEL
LIN {X 0,Y 255.071,Z 457.628,A -85,B 0,C 180,E1 -18615.642,E2 -18615.642} C_VEL
LIN {X 0,Y 254.587,Z 459.102,A -85,B 0,C 180,E1 -18617.241,E2 -18617.241} C_VEL
LIN {X 0,Y 254.058,Z 460.762,A -85,B 0,C 180,E1 -18620.446,E2 -18620.446} C_VEL
LIN {X 0,Y 253.971,Z 461.013,A -85,B 0,C 180,E1 -18622.047,E2 -18622.047} C_VEL
LIN {X 0,Y 253.991,Z 460.423,A -85,B 0,C 180,E1 -18624.961,E2 -18624.961} C_VEL
LIN {X 0,Y 254.052,Z 459.325,A -85,B 0,C 180,E1 -18626.828,E2 -18626.828} C_VEL
LIN {X 0,Y 254.141,Z 457.981,A -85,B 0,C 180,E1 -18628.415,E2 -18628.415} C_VEL
LIN {X 0,Y 254.421,Z 455.144,A -85,B 0,C 180,E1 -18630.791,E2 -18630.791} C_VEL
LIN {X 0,Y 254.924,Z 451.294,A -85,B 0,C 180,E1 -18633.161,E2 -18633.161} C_VEL
LIN {X 0,Y 255.787,Z 446.32,A -85,B 0,C 180,E1 -18635.518,E2 -18635.518} C_VEL
LIN {X 0,Y 256.845,Z 440.082,A -85,B 0,C 180,E1 -18637.863,E2 -18637.863} C_VEL
LIN {X 0,Y 258.337,Z 432.265,A -85,B 0,C 180,E1 -18640.185,E2 -18640.185} C_VEL
LIN {X 0,Y 259.904,Z 424.294,A -85,B 0,C 180,E1 -18642.097,E2 -18642.097} C_VEL
LIN {X 0,Y 261.498,Z 414.596,A -85,B 0,C 180,E1 -18643.998,E2 -18643.998} C_VEL
LIN {X 0,Y 263.02,Z 405.083,A -85,B 0,C 180,E1 -18645.498,E2 -18645.498} C_VEL
LIN {X 0,Y 264.471,Z 394.671,A -85,B 0,C 180,E1 -18646.823,E2 -18646.823} C_VEL
LIN {X 0,Y 265.915,Z 382.724,A -85,B 0,C 180,E1 -18647.992,E2 -18647.992} C_VEL
LIN {X 0,Y 266.97,Z 369.969,A -85,B 0,C 180,E1 -18648.913,E2 -18648.913} C_VEL
LIN {X 0,Y 267.664,Z 357.725,A -85,B 0,C 180,E1 -18649.509,E2 -18649.509} C_VEL
LIN {X 0,Y 269.975,Z 285.866,A -85,B 0,C 180,E1 -18651.398,E2 -18651.398} C_VEL
LIN {X 0,Y 268.757,Z 279.925,A -85,B 0,C 180,E1 -18651.691,E2 -18651.691} C_VEL
LIN {X 0,Y 261.898,Z 261.983,A -85,B 0,C 180,E1 -18652.941,E2 -18652.941} C_VEL
LIN {X 0,Y 256.679,Z 249.863,A -85,B 0,C 180,E1 -18653.939,E2 -18653.939} C_VEL
LIN {X 0,Y 256.154,Z 247.579,A -85,B 0,C 180,E1 -18654.949,E2 -18654.949} C_VEL
LIN {X 0,Y 256.098,Z 247.586,A -85,B 0,C 180,E1 -18658.578,E2 -18658.578} C_VEL
LIN {X 0,Y 256.076,Z 247.586,A -85,B 0,C 180,E1 -18661.701,E2 -18661.701} C_VEL
LIN {X 0,Y 256.084,Z 247.585,A -85,B 0,C 180,E1 -18665.193,E2 -18665.193} C_VEL
LIN {X 0,Y 256.116,Z 247.581,A -85,B 0,C 180,E1 -18667.271,E2 -18667.271} C_VEL
LIN {X 0,Y 256.057,Z 247.587,A -85,B 0,C 180,E1 -18671.203,E2 -18671.203} C_VEL
LIN {X 0,Y 256.064,Z 247.586,A -85,B 0,C 180,E1 -18675.529,E2 -18675.529} C_VEL
LIN {X 0,Y 256.056,Z 247.591,A -85,B 0,C 180,E1 -18678.796,E2 -18678.796} C_VEL
LIN {X 0,Y 256.131,Z 247.581,A -85,B 0,C 180,E1 -18682.867,E2 -18682.867} C_VEL
LIN {X 0,Y 256.069,Z 247.574,A -85,B 0,C 180,E1 -18686.707,E2 -18686.707} C_VEL
LIN {X 0,Y 256.104,Z 247.578,A -85,B 0,C 180,E1 -18690.399,E2 -18690.399} C_VEL
LIN {X 0,Y 256.189,Z 247.566,A -85,B 0,C 180,E1 -18694.861,E2 -18694.861} C_VEL
LIN {X 0,Y 256.168,Z 247.562,A -85,B 0,C 180,E1 -18699.105,E2 -18699.105} C_VEL
LIN {X 0,Y 256.301,Z 247.556,A -85,B 0,C 180,E1 -18704.085,E2 -18704.085} C_VEL
LIN {X 0,Y 256.296,Z 247.536,A -85,B 0,C 180,E1 -18708.933,E2 -18708.933} C_VEL
LIN {X 0,Y 256.47,Z 247.528,A -85,B 0,C 180,E1 -18712.125,E2 -18712.125} C_VEL
LIN {X 0,Y 256.464,Z 247.531,A -85,B 0,C 180,E1 -18716.666,E2 -18716.666} C_VEL
LIN {X 0,Y 255.952,Z 247.599,A -85,B 0,C 180,E1 -18717.979,E2 -18717.979} C_VEL
LIN {X 0,Y 254.443,Z 247.789,A -85,B 0,C 180,E1 -18719.269,E2 -18719.269} C_VEL
LIN {X 0,Y 250.661,Z 248.259,A -85,B 0,C 180,E1 -18721.862,E2 -18721.862} C_VEL
LIN {X 0,Y 249.506,Z 248.399,A -85,B 0,C 180,E1 -18723.213,E2 -18723.213} C_VEL
LIN {X 0,Y 249.374,Z 248.413,A -85,B 0,C 180,E1 -18723.673,E2 -18723.673} C_VEL
LIN {X 0,Y 249.485,Z 248.407,A -85,B 0,C 180,E1 -18728.097,E2 -18728.097} C_VEL
LIN {X 0,Y 249.252,Z 248.426,A -85,B 0,C 180,E1 -18731.383,E2 -18731.383} C_VEL
LIN {X 0,Y 249.177,Z 248.446,A -85,B 0,C 180,E1 -18736.382,E2 -18736.382} C_VEL
LIN {X 0,Y 249.08,Z 248.456,A -85,B 0,C 180,E1 -18741.519,E2 -18741.519} C_VEL
LIN {X 0,Y 249.087,Z 248.451,A -85,B 0,C 180,E1 -18745.461,E2 -18745.461} C_VEL
LIN {X 0,Y 249.039,Z 248.461,A -85,B 0,C 180,E1 -18748.975,E2 -18748.975} C_VEL
LIN {X 0,Y 249.027,Z 248.465,A -85,B 0,C 180,E1 -18752.426,E2 -18752.426} C_VEL
LIN {X 0,Y 249.047,Z 248.461,A -85,B 0,C 180,E1 -18756.343,E2 -18756.343} C_VEL
LIN {X 0,Y 248.984,Z 248.472,A -85,B 0,C 180,E1 -18760.482,E2 -18760.482} C_VEL
LIN {X 0,Y 248.992,Z 248.467,A -85,B 0,C 180,E1 -18764.882,E2 -18764.882} C_VEL
LIN {X 0,Y 249.016,Z 248.461,A -85,B 0,C 180,E1 -18767.363,E2 -18767.363} C_VEL
LIN {X 0,Y 249.052,Z 248.462,A -85,B 0,C 180,E1 -18772.198,E2 -18772.198} C_VEL
LIN {X 0,Y 249.092,Z 248.608,A -85,B 0,C 180,E1 -18774.264,E2 -18774.264} C_VEL
LIN {X 0,Y 251.146,Z 257.683,A -85,B 0,C 180,E1 -18777.88,E2 -18777.88} C_VEL
LIN {X 0,Y 252.132,Z 262.379,A -85,B 0,C 180,E1 -18779.606,E2 -18779.606} C_VEL
LIN {X 0,Y 258.562,Z 279.043,A -85,B 0,C 180,E1 -18780.857,E2 -18780.857} C_VEL
LIN {X 0,Y 262.302,Z 305.887,A -85,B 0,C 180,E1 -18782.06,E2 -18782.06} C_VEL
LIN {X 0,Y 262.849,Z 311.957,A -85,B 0,C 180,E1 -18782.296,E2 -18782.296} C_VEL
LIN {X 0,Y 260.92,Z 371.325,A -85,B 0,C 180,E1 -18783.908,E2 -18783.908} C_VEL
LIN {X 0,Y 259.98,Z 384.03,A -85,B 0,C 180,E1 -18784.533,E2 -18784.533} C_VEL
LIN {X 0,Y 258.681,Z 396.195,A -85,B 0,C 180,E1 -18785.417,E2 -18785.417} C_VEL
LIN {X 0,Y 257.048,Z 408.462,A -85,B 0,C 180,E1 -18786.644,E2 -18786.644} C_VEL
LIN {X 0,Y 255.217,Z 420.076,A -85,B 0,C 180,E1 -18788.176,E2 -18788.176} C_VEL
LIN {X 0,Y 253.289,Z 430.521,A -85,B 0,C 180,E1 -18789.918,E2 -18789.918} C_VEL
LIN {X 0,Y 251.868,Z 439.316,A -85,B 0,C 180,E1 -18791.762,E2 -18791.762} C_VEL
LIN {X 0,Y 250.231,Z 448.322,A -85,B 0,C 180,E1 -18794.107,E2 -18794.107} C_VEL
LIN {X 0,Y 248.819,Z 455.746,A -85,B 0,C 180,E1 -18796.525,E2 -18796.525} C_VEL
LIN {X 0,Y 247.784,Z 462.57,A -85,B 0,C 180,E1 -18799.376,E2 -18799.376} C_VEL
LIN {X 0,Y 247.256,Z 467.064,A -85,B 0,C 180,E1 -18801.83,E2 -18801.83} C_VEL
LIN {X 0,Y 247.019,Z 469.431,A -85,B 0,C 180,E1 -18803.465,E2 -18803.465} C_VEL
LIN {X 0,Y 246.882,Z 471.364,A -85,B 0,C 180,E1 -18805.101,E2 -18805.101} C_VEL
LIN {X 0,Y 246.88,Z 472.867,A -85,B 0,C 180,E1 -18806.736,E2 -18806.736} C_VEL
LIN {X 0,Y 246.931,Z 473.918,A -85,B 0,C 180,E1 -18808.369,E2 -18808.369} C_VEL
LIN {X 0,Y 246.983,Z 474.574,A -85,B 0,C 180,E1 -18810,E2 -18810} C_VEL
LIN {X 0,Y 246.921,Z 474.839,A -85,B 0,C 180,E1 -18811.631,E2 -18811.631} C_VEL
LIN {X 0,Y 246.856,Z 474.707,A -85,B 0,C 180,E1 -18813.264,E2 -18813.264} C_VEL
LIN {X 0,Y 247.013,Z 473.198,A -85,B 0,C 180,E1 -18816.535,E2 -18816.535} C_VEL
LIN {X 0,Y 247.285,Z 471.859,A -85,B 0,C 180,E1 -18818.17,E2 -18818.17} C_VEL
LIN {X 0,Y 247.943,Z 469.04,A -85,B 0,C 180,E1 -18820.617,E2 -18820.617} C_VEL
LIN {X 0,Y 248.94,Z 465.21,A -85,B 0,C 180,E1 -18823.053,E2 -18823.053} C_VEL
LIN {X 0,Y 250.454,Z 460.272,A -85,B 0,C 180,E1 -18825.461,E2 -18825.461} C_VEL
LIN {X 0,Y 252.375,Z 454.076,A -85,B 0,C 180,E1 -18827.838,E2 -18827.838} C_VEL
LIN {X 0,Y 254.569,Z 446.42,A -85,B 0,C 180,E1 -18830.173,E2 -18830.173} C_VEL
LIN {X 0,Y 256.7,Z 438.506,A -85,B 0,C 180,E1 -18832.114,E2 -18832.114} C_VEL
LIN {X 0,Y 259.329,Z 428.919,A -85,B 0,C 180,E1 -18833.986,E2 -18833.986} C_VEL
LIN {X 0,Y 261.842,Z 418.297,A -85,B 0,C 180,E1 -18835.646,E2 -18835.646} C_VEL
LIN {X 0,Y 264.04,Z 408.034,A -85,B 0,C 180,E1 -18836.904,E2 -18836.904} C_VEL
LIN {X 0,Y 266.188,Z 395.812,A -85,B 0,C 180,E1 -18838.053,E2 -18838.053} C_VEL
LIN {X 0,Y 267.95,Z 382.222,A -85,B 0,C 180,E1 -18838.974,E2 -18838.974} C_VEL
LIN {X 0,Y 269.122,Z 369.377,A -85,B 0,C 180,E1 -18839.532,E2 -18839.532} C_VEL
LIN {X 0,Y 271.187,Z 313.976,A -85,B 0,C 180,E1 -18840.996,E2 -18840.996} C_VEL
LIN {X 0,Y 267.974,Z 294.351,A -85,B 0,C 180,E1 -18842.074,E2 -18842.074} C_VEL
LIN {X 0,Y 261.803,Z 280.218,A -85,B 0,C 180,E1 -18843.475,E2 -18843.475} C_VEL
